# B&R Automation Studio project EFI (part 17)

### LineCtrl.typ
```iecst
TYPE
	LineControlAlarms_typ : 	STRUCT
		xAlrOvervoltage : BOOL; (*Warning alarm*)
		xAlrPrinterNoPowered : BOOL; (*Warning alarm*)
		xAlr24VdcStartSeqNoPowered : BOOL; (*Warning alarm*)
		xResetCondition : BOOL;
		xStopAlarm : BOOL;
		xCriticalAlarm : BOOL;
		xWarningAlarm : BOOL;
		xAlarmNonReseteable : BOOL;
		xAlarmReseteable : BOOL;
		xAlarmSound : BOOL;
		iReasonStop : UDINT; (*The reason to move the machine to stop*)
		iReasonWarning : UDINT;
		iReasonResetCondition : UDINT; (*The reason to active light tower's blue light*)
		iReasonCritical : UDINT; (*The reason to move the machine out of auto mode*)
	END_STRUCT;
	LineControlCommands_typ : 	STRUCT
		CalibrateCamera : BOOL;
		Print : BOOL; (*Edge commands. Reseted when managed*)
		Pause : BOOL; (*Edge commands. Reseted when managed*)
		ControlStop : BOOL; (*Edge commands. Reseted when managed*)
		Stop : BOOL; (*Edge commands. Reseted when managed*)
		Clean : BOOL; (*Edge commands. Reseted when managed*)
		EmptyBelt : BOOL; (*Edge commands. Reseted when managed*)
		PowerOff : BOOL;
		StartUp : StartUpCommands_typ;
	END_STRUCT;
	LineControlParameters_typ : 	STRUCT
		ExternalDevices : ARRAY[0..MAX_EXTERNAL_DEVICES]OF StartUpParameters_typ; (*0:Feeder||1:Primer||2:Printer||3:Dryer1||4:Dryer2||5:DryerCtrl||6:Stacker||7:UV||8:Chiller||9:Hoopers||10:OPV*)
		iNumExternalDevices : INT := 0;
		iLightTowerMode : INT; (*0: IEC Standard, 1: Customer1 request, 2: Customer2 request*)
		xBatchFeeding : BOOL; (*1: Batch feeding, 0: Continous feeding*)
		Hw : LineControlHwParameters_typ;
	END_STRUCT;
	LineControlInputs_typ : 	STRUCT
		xOvervoltageProtectionOk : BOOL;
		xPrinterPowered : BOOL;
		x24VdcStartSeqNoPowered : BOOL;
		UPSs : ARRAY[0..2]OF UPS_Inputs;
		Customer : ARRAY[0..3]OF BOOL;
	END_STRUCT;
	StartUpInputs_typ : 	STRUCT
		xPowered : BOOL; (*Some devices power management needs a second signal to switch off its branch*)
	END_STRUCT;
	StartUpOutputs_typ : 	STRUCT
		xClose : BOOL; (*Signal to active contactor coil of device's power branch*)
		xOpen : BOOL; (*Before activating the Close signal, the Open output has to be activated. A NC signal through a relay is sent as Open, so just sending close both signals are electrically sent*)
	END_STRUCT;
	LineControlOutputs_typ : 	STRUCT
		ExternalDevices : ARRAY[0..MAX_EXTERNAL_DEVICES]OF StartUpOutputs_typ; (*Signal to active contactor coil of device's power branch*)
		xRedLight : BOOL;
		xYellowLight : BOOL;
		xGreenLight : BOOL;
		xWhiteLight : BOOL;
		xBlueLight : BOOL;
		xLightReset : BOOL;
		xSound : BOOL;
		Customer : ARRAY[0..3]OF BOOL;
		Sw : LineControlOutputsForSw;
	END_STRUCT;
	StartUpCommands_typ : 	STRUCT
		xPowerOff : ARRAY[0..MAX_EXTERNAL_DEVICES]OF BOOL; (*0:Feeder||1:Primer||2:Printer||3:Dryer1||4:Dryer2||5:DryerCtrl||6:Stacker||7:UV||8:Chiller||9:Hoopers||10:OPV*)
		xPowerUp : ARRAY[0..MAX_EXTERNAL_DEVICES]OF BOOL; (*0:Feeder||1:Primer||2:Printer||3:Dryer1||4:Dryer2||5:DryerCtrl||6:Stacker||7:UV||8:Chiller||9:Hoopers||10:OPV*)
		xStartAll : BOOL;
	END_STRUCT;
	StartUpParameters_typ : 	STRUCT
		tiDelay : TIME; (*Delay to activate from the previous device*)
		xIsEngine : BOOL; (*Activate if the Power is set to de Device through a Motorized contactor*)
	END_STRUCT;
	LineControl_typ : 	STRUCT
		Commands : LineControlCommands_typ;
		Status : LineStatus_enum := LINE_NOT_POWERED;
		StatusSw : UINT := 0; (*Copy for Sw*)
		Alarms : LineControlAlarms_typ;
		Parameters : LineControlParameters_typ;
		Outputs : LineControlOutputs_typ;
		Inputs : LineControlInputs_typ;
		SubStatus : UINT; (*Substatus of Line.Status. Info useful for reports and debug*)
		StatusSummary : LineControlStatusSummarized; (*Struct to summarize different states that belongs to same process*)
		OrdersSw : LineControlOrdersSw_typ;
		Orders : LineControlOrders_typ;
	END_STRUCT;
	LineControlOutputsForSw : 	STRUCT
		xPrintOrderRequestToSw : BOOL;
		xCleanOrderRequestToSw : BOOL;
		iTimesBlockAtSafePosition : UINT; (*Counter to acknowledge how many times block has been lifted to safe position*)
	END_STRUCT;
	LineControlOrders_typ : 	STRUCT
		Preprinting : BOOL; (*Order to the printer to go to preprint position*)
	END_STRUCT;
	LineControlOrdersSw_typ : 	STRUCT
		Shutdown : BOOL;
	END_STRUCT;
	LineControlHwParameters_typ : 	STRUCT
		rMaxSpeed : REAL; (*Speed in mm/min*)
		xDoubleLineAllowed : BOOL; (*Active when allows double line printing*)
	END_STRUCT;
END_TYPE
```

### Library Logical/LineCtrl/LineCtrl

#### LineCtrlFunctions.fun
```iecst
{REDUND_ERROR} FUNCTION CuringSystemsStarted : BOOL (*TODO: Add your comment here*) (*$GROUP=User,$CAT=User,$GROUPICON=User.png,$CATICON=User.png*)
	VAR_INPUT
		CuringLed : REFERENCE TO CuringLed_typ;
	END_VAR
END_FUNCTION

{REDUND_ERROR} FUNCTION CuringSystemsReady : BOOL (*TODO: Add your comment here*) (*$GROUP=User,$CAT=User,$GROUPICON=User.png,$CATICON=User.png*)
	VAR_INPUT
		CuringLed : REFERENCE TO CuringLed_typ;
	END_VAR
END_FUNCTION

{REDUND_ERROR} FUNCTION PrinterBeltStopped : BOOL (*TODO: Add your comment here*) (*$GROUP=User,$CAT=User,$GROUPICON=User.png,$CATICON=User.png*)
	VAR_INPUT
		Belt : REFERENCE TO stBelt;
	END_VAR
END_FUNCTION

{REDUND_ERROR} FUNCTION PrinterBeltStarted : BOOL (*TODO: Add your comment here*) (*$GROUP=User,$CAT=User,$GROUPICON=User.png,$CATICON=User.png*)
	VAR_INPUT
		Belt : REFERENCE TO stBelt;
	END_VAR
END_FUNCTION

{REDUND_ERROR} FUNCTION DryerReady : BOOL (*TODO: Add your comment here*) (*$GROUP=User,$CAT=User,$GROUPICON=User.png,$CATICON=User.png*)
	VAR_INPUT
		Dryer : REFERENCE TO DryerAnc_typ;
	END_VAR
END_FUNCTION

{REDUND_ERROR} FUNCTION FeederReady : BOOL (*TODO: Add your comment here*) (*$GROUP=User,$CAT=User,$GROUPICON=User.png,$CATICON=User.png*)
	VAR_INPUT
		Feeder : REFERENCE TO Feeder_typ;
	END_VAR
END_FUNCTION

{REDUND_ERROR} FUNCTION PrimerReady : BOOL (*TODO: Add your comment here*) (*$GROUP=User,$CAT=User,$GROUPICON=User.png,$CATICON=User.png*)
	VAR_INPUT
		Primer : REFERENCE TO Primer_typ;
	END_VAR
END_FUNCTION

{REDUND_ERROR} FUNCTION SarmStopped : BOOL (*TODO: Add your comment here*) (*$GROUP=User,$CAT=User,$GROUPICON=User.png,$CATICON=User.png*)
	VAR_INPUT
		Sarm : REFERENCE TO Sarm_typ;
	END_VAR
END_FUNCTION

{REDUND_ERROR} FUNCTION SarmStarted : BOOL (*TODO: Add your comment here*) (*$GROUP=User,$CAT=User,$GROUPICON=User.png,$CATICON=User.png*)
	VAR_INPUT
		Sarm : REFERENCE TO Sarm_typ;
	END_VAR
END_FUNCTION

{REDUND_ERROR} FUNCTION SarmReady : BOOL (*TODO: Add your comment here*) (*$GROUP=User,$CAT=User,$GROUPICON=User.png,$CATICON=User.png*)
	VAR_INPUT
		Sarm : REFERENCE TO Sarm_typ;
	END_VAR
END_FUNCTION

FUNCTION EhdAdjusted : BOOL
	VAR_INPUT
		EdgeHoldDown : REFERENCE TO EdgeHoldDown_typ;
	END_VAR
END_FUNCTION

FUNCTION EhdReady : BOOL
	VAR_INPUT
		EdgeHoldDown : REFERENCE TO EdgeHoldDown_typ;
	END_VAR
END_FUNCTION

{REDUND_ERROR} FUNCTION StackerReady : BOOL (*TODO: Add your comment here*) (*$GROUP=User,$CAT=User,$GROUPICON=User.png,$CATICON=User.png*)
	VAR_INPUT
		Stacker : REFERENCE TO Stacker_typ;
	END_VAR
END_FUNCTION

{REDUND_ERROR} FUNCTION BarPositionCleaning : BOOL (*TODO: Add your comment here*) (*$GROUP=User,$CAT=User,$GROUPICON=User.png,$CATICON=User.png*)
	VAR_INPUT
		Machine : REFERENCE TO StGeneral;
	END_VAR
END_FUNCTION

{REDUND_ERROR} FUNCTION BarPositionCapped : BOOL (*TODO: Add your comment here*) (*$GROUP=User,$CAT=User,$GROUPICON=User.png,$CATICON=User.png*)
	VAR_INPUT
		Machine : REFERENCE TO StGeneral;
	END_VAR
END_FUNCTION

{REDUND_ERROR} FUNCTION JobReady : BOOL (*TODO: Add your comment here*) (*$GROUP=User,$CAT=User,$GROUPICON=User.png,$CATICON=User.png*)
	VAR_INPUT
		Machine : REFERENCE TO StGeneral;
	END_VAR
END_FUNCTION

{REDUND_ERROR} FUNCTION BarPositionReady : BOOL (*TODO: Add your comment here*) (*$GROUP=User,$CAT=User,$GROUPICON=User.png,$CATICON=User.png*)
	VAR_INPUT
		Machine : REFERENCE TO StGeneral;
	END_VAR
END_FUNCTION

{REDUND_ERROR} FUNCTION DryerStarted : BOOL (*TODO: Add your comment here*) (*$GROUP=User,$CAT=User,$GROUPICON=User.png,$CATICON=User.png*)
	VAR_INPUT
		Dryer : REFERENCE TO DryerAnc_typ;
	END_VAR
END_FUNCTION

{REDUND_ERROR} FUNCTION FeederStarted : BOOL (*TODO: Add your comment here*) (*$GROUP=User,$CAT=User,$GROUPICON=User.png,$CATICON=User.png*)
	VAR_INPUT
		Feeder : REFERENCE TO Feeder_typ;
	END_VAR
END_FUNCTION

{REDUND_ERROR} FUNCTION PrimerStarted : BOOL (*TODO: Add your comment here*) (*$GROUP=User,$CAT=User,$GROUPICON=User.png,$CATICON=User.png*)
	VAR_INPUT
		Primer : REFERENCE TO Primer_typ;
	END_VAR
END_FUNCTION

{REDUND_ERROR} FUNCTION StackerStarted : BOOL (*TODO: Add your comment here*) (*$GROUP=User,$CAT=User,$GROUPICON=User.png,$CATICON=User.png*)
	VAR_INPUT
		Stacker : REFERENCE TO Stacker_typ;
	END_VAR
END_FUNCTION

{REDUND_ERROR} FUNCTION ThicknessSensorReady : BOOL (*TODO: Add your comment here*) (*$GROUP=User,$CAT=User,$GROUPICON=User.png,$CATICON=User.png*)
	VAR_INPUT
		ThickCtrl : REFERENCE TO stThicknessCtrl_typ;
	END_VAR
END_FUNCTION

{REDUND_ERROR} FUNCTION DryerPaused : BOOL (*TODO: Add your comment here*) (*$GROUP=User,$CAT=User,$GROUPICON=User.png,$CATICON=User.png*)
	VAR_INPUT
		Dryer : REFERENCE TO DryerAnc_typ;
	END_VAR
END_FUNCTION

{REDUND_ERROR} FUNCTION PrimerPaused : BOOL (*TODO: Add your comment here*) (*$GROUP=User,$CAT=User,$GROUPICON=User.png,$CATICON=User.png*)
	VAR_INPUT
		Primer : REFERENCE TO Primer_typ;
	END_VAR
END_FUNCTION

{REDUND_ERROR} FUNCTION FeederPaused : BOOL (*TODO: Add your comment here*) (*$GROUP=User,$CAT=User,$GROUPICON=User.png,$CATICON=User.png*)
	VAR_INPUT
		Feeder : REFERENCE TO Feeder_typ;
	END_VAR
END_FUNCTION

{REDUND_ERROR} FUNCTION DryerStopped : BOOL (*TODO: Add your comment here*) (*$GROUP=User,$CAT=User,$GROUPICON=User.png,$CATICON=User.png*)
	VAR_INPUT
		Dryer : REFERENCE TO DryerAnc_typ;
	END_VAR
END_FUNCTION

{REDUND_ERROR} FUNCTION FeederStopped : BOOL (*TODO: Add your comment here*) (*$GROUP=User,$CAT=User,$GROUPICON=User.png,$CATICON=User.png*)
	VAR_INPUT
		Feeder : REFERENCE TO Feeder_typ;
	END_VAR
END_FUNCTION

{REDUND_ERROR} FUNCTION PrimerStopped : BOOL (*TODO: Add your comment here*) (*$GROUP=User,$CAT=User,$GROUPICON=User.png,$CATICON=User.png*)
	VAR_INPUT
		Primer : REFERENCE TO Primer_typ;
	END_VAR
END_FUNCTION

{REDUND_ERROR} FUNCTION StackerStopped : BOOL (*TODO: Add your comment here*) (*$GROUP=User,$CAT=User,$GROUPICON=User.png,$CATICON=User.png*)
	VAR_INPUT
		Stacker : REFERENCE TO Stacker_typ;
	END_VAR
END_FUNCTION

FUNCTION EhdStopped : BOOL
	VAR_INPUT
		EdgeHoldDown : REFERENCE TO EdgeHoldDown_typ;
	END_VAR
END_FUNCTION

{REDUND_ERROR} FUNCTION FeederNotFeeding : BOOL (*TODO: Add your comment here*) (*$GROUP=User,$CAT=User,$GROUPICON=User.png,$CATICON=User.png*)
	VAR_INPUT
		Feeder : REFERENCE TO Feeder_typ;
	END_VAR
END_FUNCTION

{REDUND_ERROR} FUNCTION OpvReady : BOOL (*TODO: Add your comment here*) (*$GROUP=User,$CAT=User,$GROUPICON=User.png,$CATICON=User.png*)
	VAR_INPUT
		OverVarnish : REFERENCE TO Opv_typ;
	END_VAR
END_FUNCTION

{REDUND_ERROR} FUNCTION OpvStarted : BOOL (*TODO: Add your comment here*) (*$GROUP=User,$CAT=User,$GROUPICON=User.png,$CATICON=User.png*)
	VAR_INPUT
		OverVarnish : REFERENCE TO Opv_typ;
	END_VAR
END_FUNCTION

FUNCTION SarmPaused : BOOL
	VAR_INPUT
		Sarm : REFERENCE TO Sarm_typ;
	END_VAR
END_FUNCTION

{REDUND_ERROR} FUNCTION OpvPaused : BOOL (*TODO: Add your comment here*) (*$GROUP=User,$CAT=User,$GROUPICON=User.png,$CATICON=User.png*)
	VAR_INPUT
		OverVarnish : REFERENCE TO Opv_typ;
	END_VAR
END_FUNCTION

{REDUND_ERROR} FUNCTION OpvStopped : BOOL (*TODO: Add your comment here*) (*$GROUP=User,$CAT=User,$GROUPICON=User.png,$CATICON=User.png*)
	VAR_INPUT
		OverVarnish : REFERENCE TO Opv_typ;
	END_VAR
END_FUNCTION

{REDUND_ERROR} FUNCTION FeederEmptied : BOOL (*TODO: Add your comment here*) (*$GROUP=User,$CAT=User,$GROUPICON=User.png,$CATICON=User.png*)
	VAR_INPUT
		Feeder : REFERENCE TO Feeder_typ;
	END_VAR
END_FUNCTION

{REDUND_ERROR} FUNCTION StackerEmptied : BOOL (*TODO: Add your comment here*) (*$GROUP=User,$CAT=User,$GROUPICON=User.png,$CATICON=User.png*)
	VAR_INPUT
		Stacker : REFERENCE TO Stacker_typ;
	END_VAR
END_FUNCTION

{REDUND_ERROR} FUNCTION OpvEmptied : BOOL (*TODO: Add your comment here*) (*$GROUP=User,$CAT=User,$GROUPICON=User.png,$CATICON=User.png*)
	VAR_INPUT
		OverVarnish : REFERENCE TO Opv_typ;
	END_VAR
END_FUNCTION

{REDUND_ERROR} FUNCTION DryerEmptied : BOOL (*TODO: Add your comment here*) (*$GROUP=User,$CAT=User,$GROUPICON=User.png,$CATICON=User.png*)
	VAR_INPUT
		Dryer : REFERENCE TO DryerAnc_typ;
	END_VAR
END_FUNCTION

{REDUND_ERROR} FUNCTION PrinterEmptied : BOOL (*TODO: Add your comment here*) (*$GROUP=User,$CAT=User,$GROUPICON=User.png,$CATICON=User.png*)
	VAR_INPUT
		ThickCtrl : REFERENCE TO stThicknessCtrl_typ;
	END_VAR
END_FUNCTION

{REDUND_ERROR} FUNCTION PrimerEmptied : BOOL (*TODO: Add your comment here*) (*$GROUP=User,$CAT=User,$GROUPICON=User.png,$CATICON=User.png*)
	VAR_INPUT
		Primer : REFERENCE TO Primer_typ;
	END_VAR
END_FUNCTION

FUNCTION SarmEmptied : BOOL
	VAR_INPUT
		Sarm : REFERENCE TO Sarm_typ;
	END_VAR
END_FUNCTION

{REDUND_ERROR} FUNCTION DryerMaxSpeed : REAL (*TODO: Add your comment here*) (*$GROUP=User,$CAT=User,$GROUPICON=User.png,$CATICON=User.png*)
	VAR_INPUT
		Dryer : REFERENCE TO DryerAnc_typ;
		Belt : REFERENCE TO stBelt;
	END_VAR
END_FUNCTION

{REDUND_ERROR} FUNCTION DryerMaxMediaLength : UINT (*TODO: Add your comment here*) (*$GROUP=User,$CAT=User,$GROUPICON=User.png,$CATICON=User.png*)
	VAR_INPUT
		Dryer : REFERENCE TO DryerAnc_typ;
		Machine : REFERENCE TO StGeneral;
	END_VAR
END_FUNCTION

{REDUND_ERROR} FUNCTION DryerMaxMediaWidth : UINT (*TODO: Add your comment here*) (*$GROUP=User,$CAT=User,$GROUPICON=User.png,$CATICON=User.png*)
	VAR_INPUT
		Dryer : REFERENCE TO DryerAnc_typ;
		Machine : REFERENCE TO StGeneral;
	END_VAR
END_FUNCTION

{REDUND_ERROR} FUNCTION FeederMaxSpeed : REAL (*TODO: Add your comment here*) (*$GROUP=User,$CAT=User,$GROUPICON=User.png,$CATICON=User.png*)
	VAR_INPUT
		Feeder : REFERENCE TO Feeder_typ;
		Belt : REFERENCE TO stBelt;
	END_VAR
END_FUNCTION

{REDUND_ERROR} FUNCTION FeederMaxMediaThickness : UINT (*TODO: Add your comment here*) (*$GROUP=User,$CAT=User,$GROUPICON=User.png,$CATICON=User.png*)
	VAR_INPUT
		Feeder : REFERENCE TO Feeder_typ;
		Machine : REFERENCE TO StGeneral;
	END_VAR
END_FUNCTION

{REDUND_ERROR} FUNCTION FeederMinMediaThickness : UINT (*TODO: Add your comment here*) (*$GROUP=User,$CAT=User,$GROUPICON=User.png,$CATICON=User.png*)
	VAR_INPUT
		Feeder : REFERENCE TO Feeder_typ;
		Machine : REFERENCE TO StGeneral;
	END_VAR
END_FUNCTION

{REDUND_ERROR} FUNCTION FeederMaxMediaLength : UINT (*TODO: Add your comment here*) (*$GROUP=User,$CAT=User,$GROUPICON=User.png,$CATICON=User.png*)
	VAR_INPUT
		Feeder : REFERENCE TO Feeder_typ;
		Machine : REFERENCE TO StGeneral;
	END_VAR
END_FUNCTION

{REDUND_ERROR} FUNCTION FeederMaxMediaWidth : UINT (*TODO: Add your comment here*) (*$GROUP=User,$CAT=User,$GROUPICON=User.png,$CATICON=User.png*)
	VAR_INPUT
		Feeder : REFERENCE TO Feeder_typ;
		Machine : REFERENCE TO StGeneral;
	END_VAR
END_FUNCTION

{REDUND_ERROR} FUNCTION PrimerMaxSpeed : REAL (*TODO: Add your comment here*) (*$GROUP=User,$CAT=User,$GROUPICON=User.png,$CATICON=User.png*)
	VAR_INPUT
		Primer : REFERENCE TO Primer_typ;
		Belt : REFERENCE TO stBelt;
	END_VAR
END_FUNCTION

{REDUND_ERROR} FUNCTION PrimerMinMediaThickness : UINT (*TODO: Add your comment here*) (*$GROUP=User,$CAT=User,$GROUPICON=User.png,$CATICON=User.png*)
	VAR_INPUT
		Primer : REFERENCE TO Primer_typ;
		Machine : REFERENCE TO StGeneral;
	END_VAR
END_FUNCTION

{REDUND_ERROR} FUNCTION PrimerMaxMediaThickness : UINT (*TODO: Add your comment here*) (*$GROUP=User,$CAT=User,$GROUPICON=User.png,$CATICON=User.png*)
	VAR_INPUT
		Primer : REFERENCE TO Primer_typ;
		Machine : REFERENCE TO StGeneral;
	END_VAR
END_FUNCTION

{REDUND_ERROR} FUNCTION PrimerMaxMediaLength : UINT (*TODO: Add your comment here*) (*$GROUP=User,$CAT=User,$GROUPICON=User.png,$CATICON=User.png*)
	VAR_INPUT
		Primer : REFERENCE TO Primer_typ;
		Machine : REFERENCE TO StGeneral;
	END_VAR
END_FUNCTION

{REDUND_ERROR} FUNCTION PrimerMaxMediaWidth : UINT (*TODO: Add your comment here*) (*$GROUP=User,$CAT=User,$GROUPICON=User.png,$CATICON=User.png*)
	VAR_INPUT
		Primer : REFERENCE TO Primer_typ;
		Machine : REFERENCE TO StGeneral;
	END_VAR
END_FUNCTION

{REDUND_ERROR} FUNCTION OvervarnishMaxSpeed : REAL (*TODO: Add your comment here*) (*$GROUP=User,$CAT=User,$GROUPICON=User.png,$CATICON=User.png*)
	VAR_INPUT
		OverVarnish : REFERENCE TO Opv_typ;
		Belt : REFERENCE TO stBelt;
	END_VAR
END_FUNCTION

{REDUND_ERROR} FUNCTION OvervarnishMaxMediaLength : UINT (*TODO: Add your comment here*) (*$GROUP=User,$CAT=User,$GROUPICON=User.png,$CATICON=User.png*)
	VAR_INPUT
		OverVarnish : REFERENCE TO Opv_typ;
		Machine : REFERENCE TO StGeneral;
	END_VAR
END_FUNCTION

{REDUND_ERROR} FUNCTION OverVarnishMaxMediaThickness : UINT (*TODO: Add your comment here*) (*$GROUP=User,$CAT=User,$GROUPICON=User.png,$CATICON=User.png*)
	VAR_INPUT
		OverVarnish : REFERENCE TO Opv_typ;
		Machine : REFERENCE TO StGeneral;
	END_VAR
END_FUNCTION

{REDUND_ERROR} FUNCTION OverVarnishMinMediaThickness : UINT (*TODO: Add your comment here*) (*$GROUP=User,$CAT=User,$GROUPICON=User.png,$CATICON=User.png*)
	VAR_INPUT
		OverVarnish : REFERENCE TO Opv_typ;
		Machine : REFERENCE TO StGeneral;
	END_VAR
END_FUNCTION

{REDUND_ERROR} FUNCTION OvervarnishMaxMediaWidth : UINT (*TODO: Add your comment here*) (*$GROUP=User,$CAT=User,$GROUPICON=User.png,$CATICON=User.png*)
	VAR_INPUT
		OverVarnish : REFERENCE TO Opv_typ;
		Machine : REFERENCE TO StGeneral;
	END_VAR
END_FUNCTION

{REDUND_ERROR} FUNCTION StackerMaxSpeed : REAL (*TODO: Add your comment here*) (*$GROUP=User,$CAT=User,$GROUPICON=User.png,$CATICON=User.png*)
	VAR_INPUT
		Stacker : REFERENCE TO Stacker_typ;
		Belt : REFERENCE TO stBelt;
	END_VAR
END_FUNCTION

{REDUND_ERROR} FUNCTION StackerMaxMediaLength : UINT (*TODO: Add your comment here*) (*$GROUP=User,$CAT=User,$GROUPICON=User.png,$CATICON=User.png*)
	VAR_INPUT
		Stacker : REFERENCE TO Stacker_typ;
		Machine : REFERENCE TO StGeneral;
	END_VAR
END_FUNCTION

{REDUND_ERROR} FUNCTION StackerMaxMediaThickness : UINT (*TODO: Add your comment here*) (*$GROUP=User,$CAT=User,$GROUPICON=User.png,$CATICON=User.png*)
	VAR_INPUT
		Stacker : REFERENCE TO Stacker_typ;
		Machine : REFERENCE TO StGeneral;
	END_VAR
END_FUNCTION

{REDUND_ERROR} FUNCTION StackerMinMediaThickness : UINT (*TODO: Add your comment here*) (*$GROUP=User,$CAT=User,$GROUPICON=User.png,$CATICON=User.png*)
	VAR_INPUT
		Stacker : REFERENCE TO Stacker_typ;
		Machine : REFERENCE TO StGeneral;
	END_VAR
END_FUNCTION

{REDUND_ERROR} FUNCTION StackerMaxMediaWidth : UINT (*TODO: Add your comment here*) (*$GROUP=User,$CAT=User,$GROUPICON=User.png,$CATICON=User.png*)
	VAR_INPUT
		Stacker : REFERENCE TO Stacker_typ;
		Machine : REFERENCE TO StGeneral;
	END_VAR
END_FUNCTION

{REDUND_ERROR} FUNCTION SarmMaxSpeed : REAL (*TODO: Add your comment here*) (*$GROUP=User,$CAT=User,$GROUPICON=User.png,$CATICON=User.png*)
	VAR_INPUT
		Sarm : REFERENCE TO Sarm_typ;
		Belt : REFERENCE TO stBelt;
	END_VAR
END_FUNCTION

{REDUND_ERROR} FUNCTION SarmMaxMediaThickness : UINT (*TODO: Add your comment here*) (*$GROUP=User,$CAT=User,$GROUPICON=User.png,$CATICON=User.png*)
	VAR_INPUT
		Sarm : REFERENCE TO Sarm_typ;
		Machine : REFERENCE TO StGeneral;
	END_VAR
END_FUNCTION

{REDUND_ERROR} FUNCTION SarmMinMediaThickness : UINT (*TODO: Add your comment here*) (*$GROUP=User,$CAT=User,$GROUPICON=User.png,$CATICON=User.png*)
	VAR_INPUT
		Sarm : REFERENCE TO Sarm_typ;
		Machine : REFERENCE TO StGeneral;
	END_VAR
END_FUNCTION

{REDUND_ERROR} FUNCTION SarmMaxMediaLength : UINT (*TODO: Add your comment here*) (*$GROUP=User,$CAT=User,$GROUPICON=User.png,$CATICON=User.png*)
	VAR_INPUT
		Sarm : REFERENCE TO Sarm_typ;
		Machine : REFERENCE TO StGeneral;
	END_VAR
END_FUNCTION

{REDUND_ERROR} FUNCTION SarmMaxMediaWidth : UINT (*TODO: Add your comment here*) (*$GROUP=User,$CAT=User,$GROUPICON=User.png,$CATICON=User.png*)
	VAR_INPUT
		Sarm : REFERENCE TO Sarm_typ;
		Machine : REFERENCE TO StGeneral;
	END_VAR
END_FUNCTION
```

#### CleaningBelt.st
```iecst
ACTION CleaningBelt:
	IF xStatusChanged THEN
		iLineStatus:=720;
	END_IF

	CASE iLineStatus OF
		720:
			gMachine.commands.CleanBelt.xStart := FALSE;
			xCleanBeltToBeExecuted := FALSE;
			IF gBeltClean.Status.State = BCLEAN_FAULT OR NOT gMachine.St.Position.xCleaning AND NOT BeltClean.Status.xCleaning THEN
				IF xPreviousIdle THEN
					gMachine.commands.xRunBelt := FALSE;
				END_IF
				xLineReady:=TRUE;
			END_IF
	END_CASE

END_ACTION
```

#### ControlStopping.st
```iecst
ACTION ControlStopping:

	IF xStatusChanged THEN
		ton_PrinterBeltInputEmpty.IN := FALSE;
		iLineStatus:=500;
	END_IF

	ton_PrinterBeltInputEmpty();

	CASE iLineStatus OF

		500:
			gMachine.commands.xClean:=FALSE;

			IF gMachine.AlSummary.xAlarmStop THEN
				Feeder.Commands.xStop:=TRUE;
				Primer.Commands.xStop:=TRUE;
				Sarm.Commands.xStop:=TRUE;
				gMachine.commands.xStop:=TRUE;
				gMachine.commands.xRunBelt:=FALSE; //This shouldnt be required, Why stop command does not stop the belt?
				StopCuringSystems;
				StopBlowers;
				iLineStatus:=506;

			ELSIF Sarm.Alarms.xCriticalAlarm THEN
				Feeder.Commands.xStop:=TRUE;
				Primer.Commands.xStop:=TRUE;
				Sarm.Commands.xStop:=TRUE;
				iLineStatus:=504;

			ELSIF Primer.Alarms.xCriticalAlarm THEN
				Feeder.Commands.xStop:=TRUE;
				Primer.Commands.xStop:=TRUE;

				iLineStatus:=503;
			ELSE
				iLineStatus:=iLineStatus+1;
			END_IF

		501:
			Feeder.Commands.xStop:=TRUE;
			iLineStatus:=iLineStatus+1;

		502:
			xFeederNotFeeding := FeederNotFeeding(ADR(Feeder));
			IF xFeederNotFeeding THEN
				Primer.Commands.xControlStop:=TRUE;
				iLineStatus:=iLineStatus+1;
			END_IF

			IF gMachine.AlSummary.xAlarmStop THEN
				Feeder.Commands.xStop:=TRUE;
				Primer.Commands.xStop:=TRUE;
				Sarm.Commands.xStop:=TRUE;
				gMachine.commands.xStop:=TRUE;
				gMachine.commands.xRunBelt:=FALSE; //This shouldnt be required, Why stop command does not stop the belt?
				StopCuringSystems;
				StopBlowers;
				iLineStatus:=506;

			ELSIF Sarm.Alarms.xCriticalAlarm THEN
				Feeder.Commands.xStop:=TRUE;
				Primer.Commands.xStop:=TRUE;
				Sarm.Commands.xStop:=TRUE;
				iLineStatus:=504;

			ELSIF Primer.Alarms.xCriticalAlarm THEN
				Feeder.Commands.xStop:=TRUE;
				Primer.Commands.xStop:=TRUE;

				iLineStatus:=503;
			END_IF

		503:
			xPrimerStopped := PrimerStopped(ADR(Primer));
			IF xPrimerStopped THEN
				Sarm.Commands.xControlStop:=TRUE;
				iLineStatus:=iLineStatus+1;
			END_IF

			IF gMachine.AlSummary.xAlarmStop THEN
				Feeder.Commands.xStop:=TRUE;
				Primer.Commands.xStop:=TRUE;
				Sarm.Commands.xStop:=TRUE;
				gMachine.commands.xStop:=TRUE;
				gMachine.commands.xRunBelt:=FALSE; //This shouldnt be required, Why stop command does not stop the belt?
				StopCuringSystems;
				StopBlowers;
				iLineStatus:=506;

			ELSIF Sarm.Alarms.xCriticalAlarm THEN
				Feeder.Commands.xStop:=TRUE;
				Primer.Commands.xStop:=TRUE;
				Sarm.Commands.xStop:=TRUE;
				iLineStatus:=504;
			END_IF

		504:
			xSarmStopped := SarmStopped(ADR(Sarm));
			IF xSarmStopped THEN
				iLineStatus:=iLineStatus+1;
			END_IF

			IF gMachine.AlSummary.xAlarmStop THEN
				Feeder.Commands.xStop:=TRUE;
				Primer.Commands.xStop:=TRUE;
				Sarm.Commands.xStop:=TRUE;
				gMachine.commands.xStop:=TRUE;
				gMachine.commands.xRunBelt:=FALSE; //This shouldnt be required, Why stop command does not stop the belt?
				StopCuringSystems;
				StopBlowers;
				iLineStatus:=506;
			END_IF

		505:
			//Timer
			tiTimeToEmpty := REAL_TO_TIME(60 * (gMachine.Pt.CT.rDistanceBeltInitToPd) / Belt.parameters.rSetPointSpeed); //Belt.parameters.rSetPointSpeed minimum value is 5m/min, cannot be 0.
			ton_PrinterBeltInputEmpty.IN := TRUE;
			ton_PrinterBeltInputEmpty.PT := tiTimeToEmpty;

			xPrinterBeltInputEmpty := ton_PrinterBeltInputEmpty.Q;

			xPrinterBeltStopped:= PrinterBeltStopped(ADR(Belt));
			IF (xPrinterBeltInputEmpty OR xFromPause) AND (xPrinterEmptied OR xPrinterBeltStopped) THEN
				StopCuringSystems;
				StopBlowers;

				EdgeHoldDown.commands.xStop := TRUE;

				iLineStatus:=iLineStatus+1;
			END_IF

			IF gMachine.AlSummary.xAlarmStop THEN
				Feeder.Commands.xStop:=TRUE;
				Primer.Commands.xStop:=TRUE;
				Sarm.Commands.xStop:=TRUE;
				gMachine.commands.xStop:=TRUE;
				gMachine.commands.xRunBelt:=FALSE; //This shouldnt be required, Why stop command does not stop the belt?
				StopCuringSystems;
				StopBlowers;
				iLineStatus:=506;
			END_IF

		506:
			xEhdStopped := EhdStopped(ADR(EdgeHoldDown));
			IF xEhdStopped AND xDryerEmptied AND xOpvEmptied THEN
				gMachine.commands.xStop:=TRUE;
				gMachine.commands.xRunBelt:=FALSE;

				EdgeHoldDown.orders.xAdjustToMedia:=FALSE;
				EdgeHoldDown.orders.xResetPosition:=TRUE;

				Dryer.Commands.xControlStop:=TRUE;
				iLineStatus:=iLineStatus+1;
			END_IF

		507:
			xDryerStopped := DryerStopped(ADR(Dryer));
			IF xDryerStopped THEN
				OverVarnish.Commands.xControlStop:=TRUE;
				iLineStatus:=iLineStatus+1;
			END_IF

		508:
			xOverVarnishStopped := OpvStopped(ADR(OverVarnish));
			IF xOverVarnishStopped THEN
				Stacker.Commands.xControlStop:=TRUE;
				iLineStatus:=iLineStatus+1;
			END_IF

		509:
			xBarsInCapPosition := BarPositionCapped(ADR(Machine));
			xEhdReady := EhdReady(ADR(EdgeHoldDown));
			IF xEhdReady AND xBarsInCapPosition THEN
				iLineStatus:=iLineStatus+1;
			END_IF

		510:
			xStackerStopped := StackerStopped(ADR(Stacker));
			IF xStackerStopped THEN
				xLineReady:=TRUE;
			END_IF

	END_CASE

END_ACTION

ACTION StopCuringSystems:

END_ACTION

ACTION StopBlowers:
	FOR iIndexTransVacuum:=1 TO MAX_LAST_TRANS_VACUUM DO
		TransVacuum[iIndexTransVacuum].Commands.xRunByLine := FALSE;
	END_FOR
END_ACTION
```

#### EmptyingBelt.st
```iecst
ACTION EmptyingBelt:

	IF xStatusChanged THEN
		ton_PrinterBeltInputEmpty.IN := FALSE;
		iLineStatus:=220;
	END_IF

	//DELOREAN-830:To lift bars up when there are no printed boards below bars, so no more curing is required
	IF (NOT ThickCtrl.status.MediaPosition.xMediaBelowMachine) THEN gMachine.commands.xAllToCap:=TRUE; END_IF

	ton_PrinterBeltInputEmpty();

	CASE iLineStatus OF
		220:
			IF xFeederEmptied THEN
				Feeder.Commands.xStop := TRUE;
				iLineStatus:=iLineStatus+1;
			END_IF

		221:
			IF xPrimerEmptied THEN
				Primer.Commands.xControlStop:=TRUE;
				iLineStatus:=iLineStatus+1;
			END_IF

		222:
			IF xSarmEmptied THEN
				Sarm.Commands.xControlStop := TRUE;
				iLineStatus:=iLineStatus+1;
			END_IF

		223:
			//Timer
			tiTimeToEmpty := REAL_TO_TIME(60 * (UINT_TO_REAL (gThicknessCtrl.parameters.Belt.iBeltPerimeterLength * 5)) / Belt.parameters.rSetPointSpeed); //Belt.parameters.rSetPointSpeed minimum value is 5m/min, cannot be 0.
			ton_PrinterBeltInputEmpty.IN := TRUE;
			ton_PrinterBeltInputEmpty.PT := tiTimeToEmpty;

			xPrinterBeltInputEmpty := ton_PrinterBeltInputEmpty.Q;
			IF xPrinterEmptied AND xPrinterBeltInputEmpty THEN
				iLineStatus:=iLineStatus+1;
			END_IF

		224:
			IF xDryerEmptied THEN
				iLineStatus:=iLineStatus+1;
			END_IF

		225:
			IF xOpvEmptied THEN
				iLineStatus:=iLineStatus+1;
			END_IF

		226:
			IF xStackerEmptied THEN
				xLineReady:=TRUE;
			END_IF

	END_CASE

END_ACTION
```

#### LineAlarms.st
```iecst
ACTION LineAlarms:

	//////////////////
	// General Alarms
	//////////////////

	//Reset Alarms//
	IF gMachine.AutoCmd.xReset THEN
		ResetAlarms;
	END_IF

	//Critical//
	//Printer Powered
	IF xLinePoweredON AND NOT Line.Inputs.xPrinterPowered THEN
		Line.Alarms.xAlrPrinterNoPowered := TRUE;
	END_IF

	//Main Supply Overvoltage
	IF NOT Line.Inputs.xOvervoltageProtectionOk THEN
		Line.Alarms.xAlrOvervoltage := TRUE;
	END_IF

	//24VDC Start Sequence Powered
	IF Line.Inputs.x24VdcStartSeqNoPowered THEN
		Line.Alarms.xAlr24VdcStartSeqNoPowered := TRUE;
	END_IF

END_ACTION

ACTION ResetAlarms:
	Line.Alarms := AlarmsReseted;
END_ACTION
```

#### LineAlarmsSummary.st
```iecst
ACTION LineAlarmsSummary:

	//////////////////
	// General Summary
	//////////////////

	//Warnings//
	iReasonWarning.0 := gMachine.AlSummary.xAnyWarning;
	iReasonWarning.1 := Feeder.Alarms.xWarningAlarm;
	iReasonWarning.2 := Primer.Alarms.xWarningAlarm;
	iReasonWarning.3 := Dryer.Alarms.xWarningAlarm;
	iReasonWarning.4 := Stacker.Alarms.xWarningAlarm;
	iReasonWarning.5 := SafetyController.Alarms.xWarningAlarm;
	iReasonWarning.6 := Sarm.Alarms.xWarningAlarm;

	Line.Alarms.xWarningAlarm :=  iReasonWarning > 0;

	//Register the reason of the warning alarm
	IF gMachine.St.Mode.xAuto AND EDGEPOS(Line.Alarms.xWarningAlarm) THEN
		Line.Alarms.iReasonWarning := iReasonWarning;
		LogWarningAlarm;
	ELSIF EDGEPOS(gMachine.St.Mode.xAuto AND NOT Line.Alarms.xWarningAlarm) THEN
		Line.Alarms.iReasonWarning := 0;
	END_IF

	//Alarms stop//
	IF gMachine.AutoCmd.xReset THEN
		iReasonStop := 0;
	END_IF

	IF (Line.Status <> LINE_STOPPED) THEN
		iReasonStop.0 := gMachine.AlSummary.xAlarmStop;
		iReasonStop.1 := Primer.Alarms.xCriticalAlarm;
		iReasonStop.2 := Line.Commands.Stop;
		iReasonStop.3 := CuringLed[1].AlSummary.xAlarmStop;
		iReasonStop.4 := CuringLed[2].AlSummary.xAlarmStop;
		iReasonStop.5 := EdgeHoldDown.AlSummary.xAlarmStop;
		iReasonStop.6 := Sarm.Alarms.xCriticalAlarm;
	END_IF

	Line.Alarms.xStopAlarm :=  iReasonStop > 0;

	//Register the reason of the Stop Alarm
	IF NOT Line.StatusSummary.xControlStopping AND EDGEPOS(Line.Alarms.xStopAlarm) THEN
		Line.Alarms.iReasonStop := iReasonStop;
		LogStopAlarm;
	ELSIF (Line.Status > LINE_STOPPED) THEN
		Line.Alarms.iReasonStop := 0;
	END_IF

	//Critical alarms//
	iReasonCritical.0 := gMachine.AlSummary.xAlarmCritical;
	iReasonCritical.1 := Dryer.Alarms.xCriticalAlarm;
	iReasonCritical.2 := Stacker.Alarms.xCriticalAlarm;
	iReasonCritical.3 := SafetyController.Alarms.xCriticalAlarm;
	iReasonCritical.4 := Line.Alarms.xAlrPrinterNoPowered;
	iReasonCritical.5 := Line.Alarms.xAlrOvervoltage;
	iReasonCritical.6 := Line.Alarms.xAlr24VdcStartSeqNoPowered;
	iReasonCritical.7 := gMachine.In.Buttons.xStop;
	iReasonCritical.8 := OverVarnish.Alarms.xCriticalAlarm;
	iReasonCritical.9 := CuringLed[1].AlSummary.xAlarmCritical;
	iReasonCritical.10 := CuringLed[2].AlSummary.xAlarmCritical;
	iReasonCritical.11 := EdgeHoldDown.AlSummary.xAlarmCritical;

	Line.Alarms.xCriticalAlarm :=  iReasonCritical > 0;

	//Register the reason of the Critical Alarm
	IF gMachine.St.Mode.xAuto AND EDGEPOS(Line.Alarms.xCriticalAlarm) THEN
		Line.Alarms.iReasonCritical := iReasonCritical;
		LogCriticalAlarm;
	ELSIF EDGEPOS(gMachine.St.Mode.xAuto AND NOT Line.Alarms.xCriticalAlarm) THEN
		Line.Alarms.iReasonCritical := 0;
	END_IF

	iReasonResetCondition.0 := (NOT Line.Alarms.xWarningAlarm) AND (Line.Alarms.iReasonWarning > 0);
	iReasonResetCondition.1 := (NOT Line.Alarms.xStopAlarm) AND (Line.Alarms.iReasonStop > 0);
	iReasonResetCondition.2 := (NOT Line.Alarms.xCriticalAlarm) AND (Line.Alarms.iReasonCritical > 0);

	Line.Alarms.xResetCondition :=  iReasonResetCondition > 0;

	xNoAlarmsActive := (NOT Line.Alarms.xCriticalAlarm) AND
						(NOT Line.Alarms.xStopAlarm);

	LightTower;
	SoundLightTower;

END_ACTION
```

#### LineCtrl.st
```iecst
PROGRAM _CYCLIC
	(* Insert code here *)
	Line ACCESS ADR(gLine);
	SafetyController ACCESS ADR (gSafetyController);
	Feeder ACCESS ADR(gFeeder);
	Primer ACCESS ADR(gPrimer);
	Sarm ACCESS ADR(gSarm);
	OverVarnish ACCESS ADR(gOverVarnish);
	Dryer ACCESS ADR(gDryerAnc);
	DryerData ACCESS ADR(gDryerRemoteData);
	Stacker ACCESS ADR(gStacker);
	Machine ACCESS ADR(gMachine);
	Belt ACCESS ADR(gBelt);
	ThickCtrl ACCESS ADR(gThicknessCtrl);
	TransVacuum ACCESS ADR(gTransVacuum);
	CuringLed ACCESS ADR(gCuringLed);
	EdgeHoldDown ACCESS ADR(gEdgeHoldDown);
	BeltClean ACCESS ADR(gBeltClean);

	//Just enter in line if gMachine controlled by line and configured the quantity of external devices
	IF NOT gMachine.Pt.xControlledByLine OR Line.Parameters.iNumExternalDevices = 0 THEN
		RETURN;
	END_IF

	Configuration;

	LineAlarms;

	LineAlarmsSummary;

	xStatusChanged := LineStatusPrevious <> Line.Status;
	IF xStatusChanged THEN xLineReady:=FALSE; iLineStatus:=0; END_IF

	xSubStatusChanged := iLineSubStatusPrevious<>iLineStatus;
	IF xSubStatusChanged THEN LogLineSubStatus;	END_IF

	LineStatusPrevious := Line.Status;
	iLineSubStatusPrevious := iLineStatus;

	//Inputs
	LineInputs;

	//External requests to line from printer (machine) or ancillaries
	LineOrders;

	CASE Line.Status OF

		LINE_NOT_POWERED:
			xLinePoweredON:=FALSE;
			//Waiting the machine to be configured
			IF Line.Parameters.iNumExternalDevices > 0 AND NOT Line.OrdersSw.Shutdown THEN
				Line.Status:=LINE_NOT_INITIALIZED;
			END_IF

		LINE_NOT_INITIALIZED:
			//xLineReady:=FALSE;
			PowerOffLineDevices;
			IF xLinePowered AND xLinePoweredOFF THEN Line.Status:=LINE_INITIALIZING; END_IF

		LINE_POWERING_OFF:
			PowerOffLineDevices;
			IF xLinePoweredOFF THEN Line.Status:=LINE_NOT_POWERED; END_IF

		LINE_INITIALIZING:
			PowerUpLineDevices;
			IF xLineReady AND xLinePoweredON THEN xLineStopped:=TRUE; Line.Status:=LINE_STOPPED; END_IF

		LINE_STOPPED:
			IF gMachine.St.Mode.xAuto THEN
				IF xLineToClean THEN
					xCleanToBeExecuted := TRUE;
					Line.Status:=LINE_PREPARING_CLEANPH;
				ELSIF xLineToCleanBelt THEN
					xCleanBeltToBeExecuted := TRUE;
					Line.Status:=LINE_PREPARING_CLEANBELT;
				ELSIF xNoAlarmsActive THEN
					Line.Status:=LINE_IDLE;
				END_IF
			END_IF

		LINE_IDLE:
			xCleanToBeExecuted:=FALSE;
			xCleanBeltToBeExecuted:=FALSE;
			xPreviousIdle:=TRUE;

			IF Line.OrdersSw.Shutdown THEN
				Line.Status:=LINE_POWERING_OFF;
			END_IF

			IF xLineToPrint AND xNoAlarmsActive THEN
				Line.Status:=LINE_PREPARING_PRINT;
			ELSIF xLineToClean THEN
				xCleanToBeExecuted := TRUE;
				Line.Status:=LINE_PREPARING_CLEANPH;
			ELSIF xLineToCleanBelt AND ThickCtrl.status.Belt.xBeltEmpty THEN
				xCleanBeltToBeExecuted := TRUE;
				Line.Status:=LINE_PREPARING_CLEANBELT;
			ELSIF xLineToEmptyBelt THEN
				Line.Status:=LINE_PREPARING_EMPTYBELT;
			END_IF

		LINE_PREPARING_EMPTYBELT:
			xLineStopped:=FALSE;
			PreparingEmptyBelt;
			IF xLineReady THEN Line.Status:=LINE_STARTING_EMPTYBELT; END_IF

		LINE_STARTING_EMPTYBELT:
			StartingEmptyBelt;
			IF xLineReady THEN Line.Status:=LINE_BELT_EMPTYING; END_IF

		LINE_BELT_EMPTYING:
			//To finish this process automatically when line is full emptied
			EmptyingBelt;
			IF xLineReady THEN Line.Status:=LINE_CONTROLLED_STOP; END_IF

		LINE_PREPARING_PRINT:
			xLineStopped:=FALSE;
			xPreviousPrinting:=FALSE;
			PreparingPrint;
			IF xLineReady THEN Line.Status:=LINE_STARTING_PRINTING; END_IF

		LINE_STARTING_PRINTING:
			StartingPrinting;
			IF xLineReady THEN Line.Status:=LINE_PRINTING; END_IF

		LINE_PRINTING:
			xPreviousIdle:=FALSE;
			IF xLineToPause OR xLineToClean OR xLineToCleanBelt THEN
				IF xLineToClean THEN
					xPreviousPrinting:=TRUE;
					xCleanToBeExecuted := TRUE;
				ELSIF xLineToCleanBelt THEN
					xPreviousPrinting:=TRUE;
					xCleanBeltToBeExecuted := TRUE;
				END_IF
				Line.Status:=LINE_PAUSING;
			END_IF

		LINE_PAUSING:
			xPreviousPausing:=FALSE;
			Pausing;
			IF xLineToClean THEN
				xCleanToBeExecuted := TRUE;
			END_IF

			IF xLineToPrint THEN
				Line.Status:=LINE_PREPARING_PRINT;
			ELSIF xLineReady THEN
				Line.Status:=LINE_PAUSED;
			END_IF

		LINE_PAUSED:
			IF xLineToPrint THEN
				Line.Status:=LINE_PREPARING_PRINT;
			ELSIF xLineToClean THEN
				xCleanToBeExecuted := TRUE;
				xPreviousPausing:=TRUE;
				Line.Status:=LINE_PREPARING_CLEANPH;
			ELSIF xLineToCleanBelt THEN
				xCleanBeltToBeExecuted := TRUE;
				xPreviousPausing:=TRUE;
				Line.Status:=LINE_PREPARING_CLEANBELT;
			END_IF

		LINE_PREPARING_CLEANPH:
			PreparingCleaningPH;
			IF xLineReady THEN Line.Status:=LINE_STARTING_CLEANINGPH; END_IF

		LINE_PREPARING_CLEANBELT:
			PreparingCleaningBelt;
			IF xLineReady THEN Line.Status:=LINE_STARTING_CLEANINGBELT; END_IF

		LINE_STARTING_CLEANINGPH:
			xCleanToBeExecuted := FALSE;
			StartingCleaningPH;
			IF xLineReady THEN Line.Status:=LINE_CLEANINGPH; END_IF

		LINE_STARTING_CLEANINGBELT:
			xCleanBeltToBeExecuted := FALSE;
			StartingCleaningBelt;
			IF xLineReady THEN Line.Status:=LINE_CLEANINGBELT; END_IF

		LINE_CLEANINGPH:
			IF NOT gMachine.St.Position.xCleaning AND NOT BeltClean.Status.xCleaning THEN
				Line.Status:=LINE_CLEANED;
			END_IF

		LINE_CLEANINGBELT:
			CleaningBelt;
			IF xLineReady THEN
				Line.Status:=LINE_CLEANED;
			END_IF

		LINE_CLEANED:
			IF xPreviousPrinting THEN
				Line.Status:=LINE_PREPARING_PRINT;
			ELSIF xPreviousIdle THEN
				Line.Status:=LINE_IDLE;
			ELSIF xPreviousPausing THEN
				Line.Status:=LINE_PAUSING;
			ELSE
				Line.Status:=LINE_STOPPED;
			END_IF

		LINE_CONTROLLED_STOP:
			xCleanBeltToBeExecuted := FALSE;
			ControlStopping;
			IF xLineReady THEN xLineStopped:=TRUE; Line.Status:=LINE_STOPPED; END_IF

		LINE_ERROR:
			Stopping;
			IF xLineReady THEN xLineStopped:=TRUE; Line.Status:=LINE_STOPPED; END_IF

	END_CASE

	StatusSw;
	IF xStatusChanged THEN LogLineSwStatus; END_IF

	//Line state summaries
	IF Line.Status<>LINE_NOT_INITIALIZED AND Line.Status<>LINE_INITIALIZING THEN
		IF NOT (xLinePowered AND xLinePoweredON) THEN
			StopAllLineDevices;
			Line.Status:=LINE_NOT_INITIALIZED;
		ELSIF (NOT xLineStopped) THEN
			IF (NOT gMachine.St.Mode.xAuto) THEN
				Line.Status:=LINE_ERROR;
			ELSIF Line.Alarms.xCriticalAlarm THEN
				Line.Status:=LINE_ERROR;
			ELSIF Line.Alarms.xStopAlarm THEN
				Line.Status:=LINE_CONTROLLED_STOP;
			END_IF
		ELSE
			IF NOT gMachine.St.Mode.xAuto THEN
				Line.Status := LINE_STOPPED;
			END_IF
		END_IF
	END_IF

	//Store the history of the status to easy the debug
	IF Line.Status<>StateHistory[0] THEN
		FOR iIndexHistory:=iHistoryLines TO 1 BY -1 DO
			StateHistory[iIndexHistory]:=StateHistory[iIndexHistory-1];
		END_FOR
		StateHistory[0]:=Line.Status;
	END_IF

	//Previous states
	xFromPause := StateHistory[1] = LINE_PAUSED;

	//Resetting local status variables
	IF EDGEPOS(Line.Alarms.xStopAlarm OR Line.Alarms.xCriticalAlarm) OR Line.StatusSummary.xIdle THEN
		//xPreviousIdle := FALSE;
		xPreviousPausing := FALSE;
		xPreviousPrinting := FALSE;
	END_IF

	//Logging commands
	IF EDGEPOS(Line.Commands.Print) THEN LogPrintCommand; END_IF
	IF EDGEPOS(Line.Commands.Pause) THEN LogPauseCommand; END_IF
	IF EDGEPOS(Line.Commands.Stop) THEN LogStopCommand; END_IF
	IF EDGEPOS(Line.Commands.Clean) THEN LogCleanCommand; END_IF
	IF EDGEPOS(Line.Commands.EmptyBelt) THEN LogEmptyBeltCommand; END_IF

	//Logging buttons
	IF EDGEPOS(gMachine.In.Buttons.xStart) THEN LogStartButton; END_IF
	IF EDGEPOS(gMachine.In.Buttons.xStop) THEN LogStopButton; END_IF

	Line.SubStatus := iLineStatus;

	//Outputs
	LineOutputs;

	//Line commands
	Line.Commands := ResetedLineCommands;

	//Line summary
	Line.StatusSummary.xStopped 		:= Line.Status=LINE_STOPPED OR Line.Status=LINE_IDLE;
	Line.StatusSummary.xErrorStopping 	:= Line.Status=LINE_ERROR;
	Line.StatusSummary.xControlStopping := Line.Status=LINE_CONTROLLED_STOP;
	Line.StatusSummary.xCleaning 		:= (Line.Status=LINE_PREPARING_CLEANPH) OR (Line.Status=LINE_STARTING_CLEANINGPH) OR (Line.Status=LINE_CLEANINGPH) OR (Line.Status=LINE_CLEANED);
	Line.StatusSummary.xCleaningBelt	:= (Line.Status=LINE_PREPARING_CLEANBELT) OR (Line.Status=LINE_STARTING_CLEANINGBELT) OR (Line.Status=LINE_CLEANINGBELT);
	Line.StatusSummary.xPausing 		:= (Line.Status=LINE_PAUSING) OR (Line.Status=LINE_PAUSED);
	Line.StatusSummary.xPrinting 		:= (Line.Status=LINE_PREPARING_PRINT) OR (Line.Status=LINE_STARTING_PRINTING) OR (Line.Status=LINE_PRINTING);
	Line.StatusSummary.xEmptyingBelts 	:= (Line.Status=LINE_PREPARING_EMPTYBELT) OR (Line.Status=LINE_STARTING_EMPTYBELT) OR (Line.Status=LINE_BELT_EMPTYING);
	Line.StatusSummary.xIdle	 		:= Line.Status=LINE_IDLE;

	xFeederEmptied := FeederEmptied(ADR(Feeder));
	xPrimerEmptied := PrimerEmptied(ADR(Primer));
	xSarmEmptied := SarmEmptied(ADR(Sarm));
	xPrinterEmptied := PrinterEmptied(ADR(ThickCtrl));
	xDryerEmptied := DryerEmptied(ADR(Dryer));
	xOpvEmptied := OpvEmptied(ADR(OverVarnish));
	xStackerEmptied := StackerEmptied(ADR(Stacker));
	Line.StatusSummary.xLineEmpty := xFeederEmptied AND xPrimerEmptied AND xSarmEmptied AND xPrinterEmptied AND xDryerEmptied AND xOpvEmptied AND xStackerEmptied; //Status added to let sw know whether line is empty

END_PROGRAM
```

#### LineOrders.st
```iecst
ACTION LineOrders:

	//Line to clean orders
	IF gMachine.St.Cleaning.xCleanRequestToLine THEN
		xCleanRequestToLine := TRUE;
	ELSE
		xCleanRequestToLine := FALSE;
	END_IF

	iReasonLineToClean.0 := Line.Commands.Clean;
	iReasonLineToClean.1 := xCleanRequestToLine;
	iReasonLineToClean.2 := xCleanToBeExecuted;

	xLineToClean := iReasonLineToClean>0;

	iReasonLineToCleanBelt.0 := BeltClean.Status.xCleanRequested;
	iReasonLineToCleanBelt.1 := xCleanBeltToBeExecuted;

	xLineToCleanBelt := iReasonLineToCleanBelt >0 AND gBeltClean.Status.State <> BCLEAN_FAULT;

	IF EdgeHoldDown.status.xEnabled AND (rEhdBarsHeighSp <> EdgeHoldDown.parameters.rBarsHeighSp) THEN
		xEhdRequestToPause := TRUE;

	ELSIF EDGENEG(Line.StatusSummary.xPausing) THEN
		xEhdRequestToPause := FALSE;
	END_IF

	//Line to pause orders
	iReasonLineToPause.0 := Line.Commands.Pause;
	iReasonLineToPause.1 := gMachine.In.Buttons.xStart;
	iReasonLineToPause.2 := Feeder.Alarms.xCriticalAlarm;
	iReasonLineToPause.3 := NOT gMachine.St.xRobotReadyToPrint AND NOT gCamera.OrdersSw.xCalibration;
	iReasonLineToPause.4 := EDGEPOS(xEhdRequestToPause);

	//Saving previous ehd heigh setpoint
	rEhdBarsHeighSp := EdgeHoldDown.parameters.rBarsHeighSp;

	//Line to print orders
	iReasonLineToPrint.0 := Line.Commands.Print;
	iReasonLineToPrint.1 := gMachine.In.Buttons.xStart AND gMachine.St.xRobotReadyToPrint AND Line.Status=LINE_PAUSED;
	iReasonLineToPrint.2 := xEhdRequestToPause AND (EdgeHoldDown.parameters.rBlockPosition>=EdgeHoldDown.status.rBlockPrePrintingPosition) AND Line.Status=LINE_PAUSED; //NOZOMITWO-2420

	//[RGP]DELOREAN-972
	//User request to print
	iReasonRequestLineToPrint.0 := tonLineStartButton.Q AND gMachine.parSw.UI.xStartPrintButtonActive;
	xLineRequestToPrintToSw:=iReasonRequestLineToPrint>0;

	//Empty belt
	iReasonLineToEmptyBelt.0 := Line.Commands.EmptyBelt;

	//To manage that these internal orders are not active at the same time
	IF iReasonLineToPause>0 AND Line.StatusSummary.xPrinting THEN
		xLineToPause := TRUE;

	ELSIF iReasonLineToPrint>0 THEN
		xLineToPrint := TRUE;

	ELSIF iReasonLineToEmptyBelt>0 THEN
		xLineToEmptyBelt := TRUE;

	ELSE
		xLineToPause := FALSE;
		xLineToPrint := FALSE;
		xLineToEmptyBelt := FALSE;
	END_IF

	//EHD
	//To send ehd to resting position when entering idle. So maybe controlled stop has not been executed properly
	IF EDGEPOS(Line.StatusSummary.xIdle) THEN
		EdgeHoldDown.orders.xResetPosition := TRUE;
	ELSIF EdgeHoldDown.status.xInRestingPosition THEN
		EdgeHoldDown.orders.xResetPosition := FALSE;
	END_IF

	//Primer NOZOMITWO-2264
	Primer.Orders.xEnablePriming := NOT Line.StatusSummary.xEmptyingBelts OR NOT Machine.St.HwData.xIsWater;

	//OPV NOZOMITWO-2264
	OverVarnish.Orders.xEnablePriming := NOT Line.StatusSummary.xEmptyingBelts OR NOT Machine.St.HwData.xIsWater;

	//Preprinting position
	ton_FeederEmpty(IN:=(NOT Feeder.Status.Device.xFeeding), PT:=T#20S);
	ton_PrimerBeltEmpty(IN:=((Primer.Inputs.Comms.xBeltEmpty OR NOT Primer.ParSw.xEnabled OR NOT Primer.Parameters.xInstalled) AND Belt.states.xRuningBelt), PT:=T#20S);
	ton_SarmBeltEmpty(IN:=((Sarm.Status.xBeltEmpty OR NOT Sarm.ParSw.xEnabled OR NOT Sarm.Parameters.xInstalled) AND Belt.states.xRuningBelt), PT:=T#20S);

	IF NOT Feeder.ParSw.xEnabled AND NOT Primer.ParSw.xEnabled AND NOT Sarm.ParSw.xEnabled THEN
		//No ancillaries installed before the printer are enabled in remote mode
		Line.Orders.Preprinting := FALSE;

	ELSE
		Line.Orders.Preprinting := 	ton_FeederEmpty.Q AND
									ton_PrimerBeltEmpty.Q AND
									ton_SarmBeltEmpty.Q AND
									(ThickCtrl.status.Belt.xBeltEmpty AND Belt.states.xRuningBelt);
	END_IF

	//SafetyController.Orders.xDisableReadBlock := NOT (gPLC.Internal.Blink_2s.Out AND gPLC.Internal.Blink_1s.Out);
	Feeder.Orders.xDisableReadBlock := NOT (gPLC.Internal.Blink_2s.Out AND gPLC.Internal.Blink_1s.Out) OR NOT Feeder.ParSw.xEnabled;
	Primer.Orders.xDisableReadBlock := NOT (NOT gPLC.Internal.Blink_2s.Out AND gPLC.Internal.Blink_1s.Out) OR NOT Primer.ParSw.xEnabled;
	Sarm.Orders.xDisableReadBlock := NOT (NOT gPLC.Internal.Blink_2s.Out AND gPLC.Internal.Blink_1s.Out) OR NOT Sarm.ParSw.xEnabled;
	OverVarnish.Orders.xDisableReadBlock := NOT (gPLC.Internal.Blink_2s.Out AND NOT gPLC.Internal.Blink_1s.Out) OR NOT OverVarnish.ParSw.xEnabled;
	Stacker.Orders.xDisableReadBlock := NOT (NOT gPLC.Internal.Blink_2s.Out AND NOT gPLC.Internal.Blink_1s.Out) OR NOT Stacker.ParSw.xEnabled;

END_ACTION
```

#### Pausing.st
```iecst
ACTION Pausing:

	IF xStatusChanged THEN
		ton_PrinterBeltInputEmpty.IN := FALSE;
		iLineStatus:=330;
	END_IF

	ton_PrinterBeltInputEmpty();

	CASE iLineStatus OF
		330:
			Feeder.Commands.xPause:=TRUE;
			xFeederPaused := FeederPaused(ADR(Feeder)) OR FeederStopped(ADR(Feeder));
			IF xFeederPaused THEN
				iLineStatus:=iLineStatus+1;
			END_IF

		331:
			Primer.Commands.xPause:=TRUE;
			xPrimerPaused := PrimerPaused(ADR(Primer));
			IF xPrimerPaused THEN
				iLineStatus:=iLineStatus+1;
			END_IF

		332:
			Sarm.Commands.xPause:=TRUE;
			xSarmPaused := SarmPaused(ADR(Sarm));
			IF xSarmPaused THEN
				iLineStatus:=iLineStatus+1;
			END_IF

		333:
			//Timer
			tiTimeToEmpty := REAL_TO_TIME(60 * (gMachine.Pt.CT.rDistanceBeltInitToPd) / Belt.parameters.rSetPointSpeed); //Belt.parameters.rSetPointSpeed minimum value is 5m/min, cannot be 0.
			ton_PrinterBeltInputEmpty.IN := TRUE;
			ton_PrinterBeltInputEmpty.PT := tiTimeToEmpty;

			xPrinterBeltInputEmpty := ton_PrinterBeltInputEmpty.Q;
			IF xPrinterBeltInputEmpty AND xPrinterEmptied THEN
				Dryer.Commands.xPause:=TRUE;
				OverVarnish.Commands.xPause:=TRUE;
				iLineStatus:=iLineStatus+1;
			END_IF

		334:
			xDryerPaused := DryerPaused(ADR(Dryer));
			IF xDryerPaused  THEN
				iLineStatus:=iLineStatus+1;
			END_IF

		335:
			xOverVarnishPaused := OpvPaused(ADR(OverVarnish));
			IF xOverVarnishPaused THEN
				xLineReady:=TRUE;
			END_IF

	END_CASE

END_ACTION
```

#### PowerUpLineDevices.st
```iecst
ACTION PowerUpLineDevices:

	IF xStatusChanged THEN
		iLineStatus:=110;
		iIndexPower:=0;
	END_IF

	CASE iLineStatus OF

		110:
			//Timer
			ton_DelayPowerOn.IN := TRUE;
			ton_DelayPowerOn.PT:= Line.Parameters.ExternalDevices[iIndexPower].tiDelay;
			ton_DelayPowerOn();

			IF Line.Parameters.ExternalDevices[iIndexPower].xIsEngine THEN
				//Activate the first output signal
				Line.Outputs.ExternalDevices[iIndexPower].xOpen:=TRUE;

				IF ton_DelayPowerOn.Q THEN
					//Activate second signal when motorized contactor is loaded
					Line.Outputs.ExternalDevices[iIndexPower].xClose:=TRUE;

					//Go to next
					ResetPowerOnTimerAndNext;
				END_IF

			ELSE
				IF ton_DelayPowerOn.Q THEN
					//Activate both outputs if it is not Motorized contactor
					Line.Outputs.ExternalDevices[iIndexPower].xClose:=TRUE;
					Line.Outputs.ExternalDevices[iIndexPower].xOpen:=TRUE;

					//Go to next
					ResetPowerOnTimerAndNext;
				END_IF
			END_IF
			iLastIndexPower := iIndexPower;

		111:

			IF iIndexPower<=Line.Parameters.iNumExternalDevices THEN
				//If the Index is not the last one, repeate the timer to activate next one
				iLineStatus:=110;
			ELSE
				iLineStatus:=iLineStatus+1;
			END_IF

		112:
			xLinePoweredON := TRUE;
			xLineReady:=TRUE;

	END_CASE

END_ACTION

ACTION ResetPowerOnTimerAndNext:

	//Reset timer
	ton_DelayPowerOn(IN:=FALSE);
	iIndexPower:=iIndexPower+1;
	iLineStatus:=iLineStatus+1;

END_ACTION
```

#### PreparingCleaningBelt.st
```iecst
ACTION PreparingCleaningBelt:

	IF xStatusChanged THEN
		iLineStatus:=700;
	END_IF

	CASE iLineStatus OF
		700:
			IF gBeltClean.Status.State = BCLEAN_FAULT THEN
				xLineReady := TRUE;
			ELSE //IF gThicknessCtrl.status.Belt.xBeltEmpty THEN
				IF xPreviousIdle AND gThicknessCtrl.status.Belt.xBeltEmpty THEN
					gMachine.commands.xRunBelt := TRUE;
				END_IF
				IF gBelt.states.xRuningBelt THEN
					gMachine.commands.CleanBelt.xStart := TRUE;
					xLineReady:=TRUE;
				END_IF
			END_IF

	END_CASE

END_ACTION
```

#### PreparingEmptyBelt.st
```iecst
ACTION PreparingEmptyBelt:

	IF xStatusChanged THEN
		iLineStatus:=200;
	END_IF

	ton_StackerCleanBelts.IN:=Stacker.Outputs.xCleanBelts;
	ton_StackerCleanBelts.PT:=T#2S;
	ton_StackerCleanBelts();

	CASE iLineStatus OF
		200:
			StartBlowers;
			IF ton_StackerCleanBelts.Q OR NOT Stacker.ParSw.xEnabled THEN
				IF (gMachine.St.HwData.xIsWater OR NOT ThickCtrl.status.MediaPosition.xMediaBelowMachine) THEN
					gMachine.commands.xAllToCap := TRUE;
					Stacker.Commands.xPrepare := TRUE;

					xBarsInCapPosition := BarPositionCapped(ADR(Machine));
					IF xBarsInCapPosition THEN iLineStatus:=iLineStatus+1; END_IF

				ELSE
					gMachine.commandsSw.xToNormal_GI := TRUE;
					IF gMachine.St.AutoMode.xProduction THEN
						gMachine.commandsSw.xToNormal_GI := FALSE; //TOREVIEW: This should be an internal command, not something coming from Comms
						gMachine.commands.xAllToPrint:=TRUE;
						Stacker.Commands.xPrepare := TRUE;

						xBarsInPrintingPosition := BarPositionReady(ADR(Machine));
						IF xBarsInPrintingPosition THEN iLineStatus:=iLineStatus+1; END_IF
					END_IF
				END_IF
			END_IF

		201:
			//Waiting stacker and evaluate which next object must be prepared
			xStackerReady := StackerReady(ADR(Stacker));
			IF xStackerReady THEN
				iLineStatus:=iLineStatus+1;
			END_IF

		202:
			OverVarnish.Commands.xPrepare:=TRUE;
			xOverVarnishReady:=OpvReady(ADR(OverVarnish));
			IF xOverVarnishReady THEN
				iLineStatus:=iLineStatus+1;
			END_IF

		203:
			IF (Dryer.ParSw.xEnableArcLamp OR Dryer.ParSw.xEnableNIR) THEN
				Dryer.Commands.xBelEmpty := TRUE;
			ELSE
				Dryer.Commands.xStartTransport:=TRUE;
			END_IF
			iLineStatus:=iLineStatus+1;

		204:
			IF Dryer.Status.CtrlStatus = DRYERCTRL_MOVING AND (Dryer.ParSw.xEnableArcLamp OR Dryer.ParSw.xEnableNIR) THEN
				Dryer.Commands.xPrepare:=TRUE;
			END_IF
			xDryerReady := DryerReady(ADR(Dryer));
			IF xDryerReady THEN xLineReady:=TRUE; END_IF

	END_CASE

END_ACTION

ACTION StartBlowers:
	FOR iIndexTransVacuum:=1 TO MAX_LAST_TRANS_VACUUM DO
		TransVacuum[iIndexTransVacuum].Commands.xRunByLine := TRUE;
	END_FOR
END_ACTION
```

#### StartingEmptyBelt.st
```iecst
ACTION StartingEmptyBelt:

	IF xStatusChanged THEN
		iLineStatus:=210;
	END_IF

	CASE iLineStatus OF
		210:
			Stacker.Commands.xStart:=TRUE;
			iLineStatus:=iLineStatus+1;

		211:
			xStackerStarted:=StackerStarted(ADR(Stacker));
			IF xStackerStarted THEN
				OverVarnish.Commands.xStart:=TRUE;
				iLineStatus:=iLineStatus+1;
			END_IF

		212:
			xOverVarnishStarted:=OpvStarted(ADR(OverVarnish));
			IF xOverVarnishStarted THEN
				Dryer.Commands.xStart:=TRUE;
				iLineStatus:=iLineStatus+1;
			END_IF

		213:
			xDryerStarted:=DryerStarted(ADR(Dryer));
			xThicknessSensorReady := ThicknessSensorReady(ADR(ThickCtrl));
			IF xThicknessSensorReady AND xDryerStarted THEN
				gMachine.commands.xRunBelt := TRUE;
				iLineStatus:=iLineStatus+1;
			END_IF

		214:
			xPrinterBeltStarted:= PrinterBeltStarted(ADR(Belt));
			IF xPrinterBeltStarted THEN
				Sarm.Commands.xStart:=TRUE;
				iLineStatus:=iLineStatus+1;
			END_IF

		215:
			xSarmStarted := SarmStarted(ADR(Sarm));
			IF xSarmStarted THEN
				Primer.Commands.xPrepare:=TRUE;
				iLineStatus:=iLineStatus+1;
			END_IF

		216:
			xPrimerReady:=PrimerReady(ADR(Primer));
			IF xPrimerReady THEN
				Feeder.Commands.xPrepare:=TRUE;
				iLineStatus:=iLineStatus+1;
			END_IF

		217:
			xFeederReady:=FeederReady(ADR(Feeder));
			IF xFeederReady THEN
				xLineReady:=TRUE;
			END_IF

	END_CASE

END_ACTION
```

#### StatusSw.st
```iecst
ACTION StatusSw:
	CASE Line.Status OF
		LINE_NOT_POWERED: Line.StatusSw:= 999;
		LINE_POWERING_OFF: Line.StatusSw:= 60;
		LINE_ERROR:	Line.StatusSw:= 2;
		LINE_PREPARING_EMPTYBELT: Line.StatusSw:= 20;
		LINE_PREPARING_PRINT: Line.StatusSw:= 30;
		LINE_PREPARING_CLEANPH: Line.StatusSw:= 40;
		LINE_PREPARING_CLEANBELT: Line.StatusSw:= 70;
		LINE_STARTING_PRINTING: Line.StatusSw:= 31;
		LINE_STARTING_CLEANINGPH: Line.StatusSw:= 41;
		LINE_STARTING_CLEANINGBELT: Line.StatusSw:= 71;
		LINE_BELT_EMPTYING:	Line.StatusSw:= 22;
		LINE_CLEANED:	Line.StatusSw:= 43;
		LINE_STARTING_EMPTYBELT: Line.StatusSw:= 21;
		LINE_IDLE:	Line.StatusSw:= 11;
		LINE_PRINTING:	Line.StatusSw:= 32;
		LINE_PAUSING:	Line.StatusSw:= 33;
		LINE_PAUSED:	Line.StatusSw:= 34;
		LINE_CLEANINGPH:	Line.StatusSw:= 42;
		LINE_CLEANINGBELT:	Line.StatusSw:= 72;
		LINE_CONTROLLED_STOP:	Line.StatusSw:= 50;
		LINE_STOPPED:	Line.StatusSw:= 10;
		LINE_NOT_INITIALIZED:	Line.StatusSw:= 0;
		LINE_INITIALIZING:	Line.StatusSw:= 5;
	END_CASE

END_ACTION
```

#### SystemsLimits.st
```iecst
FUNCTION FeederMaxMediaWidth
	IF Feeder.ParSw.xEnabled THEN FeederMaxMediaWidth:= Feeder.Parameters.Hw.iMaxMediaWidth; ELSE FeederMaxMediaWidth:= Machine.Pt.Hw.iWidth; END_IF
END_FUNCTION

FUNCTION FeederMaxMediaLength
	IF Feeder.ParSw.xEnabled THEN FeederMaxMediaLength:= Feeder.Parameters.Hw.iMaxMediaLength; ELSE FeederMaxMediaLength:= Machine.parSw.Hw.iMaxMediaLength; END_IF
END_FUNCTION

FUNCTION FeederMaxMediaThickness
	IF Feeder.ParSw.xEnabled THEN FeederMaxMediaThickness:= Feeder.Parameters.Hw.iMaxMediaThickness; ELSE FeederMaxMediaThickness:= REAL_TO_UINT(Machine.Pt.CT.rMaxTicknessMedia*10); END_IF
END_FUNCTION

FUNCTION FeederMinMediaThickness
	IF Feeder.ParSw.xEnabled THEN FeederMinMediaThickness:= Feeder.Parameters.Hw.iMinMediaThickness; ELSE FeederMinMediaThickness:= REAL_TO_UINT(Machine.Pt.CT.rMinTicknessMedia*10); END_IF
END_FUNCTION

FUNCTION FeederMaxSpeed
	IF Feeder.Parameters.xInstalled THEN FeederMaxSpeed:= Feeder.Parameters.Hw.rMaxSpeed; ELSE FeederMaxSpeed:= Belt.states.Hw.rMaxSpeed; END_IF
END_FUNCTION

FUNCTION PrimerMaxMediaWidth
	IF Primer.ParSw.xEnabled THEN PrimerMaxMediaWidth:= Primer.Parameters.Hw.iMaxMediaWidth; ELSE PrimerMaxMediaWidth:= Machine.Pt.Hw.iWidth; END_IF
END_FUNCTION

FUNCTION PrimerMaxMediaLength
	IF Primer.ParSw.xEnabled THEN PrimerMaxMediaLength:= Primer.Parameters.Hw.iMaxMediaLength; ELSE PrimerMaxMediaLength:= Machine.parSw.Hw.iMaxMediaLength; END_IF
END_FUNCTION

FUNCTION PrimerMaxMediaThickness
	IF Primer.ParSw.xEnabled THEN PrimerMaxMediaThickness:= Primer.Parameters.Hw.iMaxMediaThickness; ELSE PrimerMaxMediaThickness:= REAL_TO_UINT(Machine.Pt.CT.rMaxTicknessMedia*10); END_IF
END_FUNCTION

FUNCTION PrimerMinMediaThickness
	IF Primer.ParSw.xEnabled THEN PrimerMinMediaThickness:= Primer.Parameters.Hw.iMinMediaThickness; ELSE PrimerMinMediaThickness:= REAL_TO_UINT(Machine.Pt.CT.rMinTicknessMedia*10); END_IF
END_FUNCTION

FUNCTION PrimerMaxSpeed
	IF Primer.Parameters.xInstalled THEN PrimerMaxSpeed:= Primer.Parameters.Hw.rMaxSpeed; ELSE PrimerMaxSpeed:= Belt.states.Hw.rMaxSpeed; END_IF
END_FUNCTION

FUNCTION DryerMaxMediaWidth
	IF Dryer.ParSw.xEnabled THEN DryerMaxMediaWidth:= Dryer.Parameters.Hw.iMaxMediaWidth; ELSE DryerMaxMediaWidth:= Machine.Pt.Hw.iWidth; END_IF
END_FUNCTION

FUNCTION DryerMaxMediaLength
	IF Dryer.ParSw.xEnabled THEN DryerMaxMediaLength:= Dryer.Parameters.Hw.iMaxMediaLength; ELSE DryerMaxMediaLength:= Machine.parSw.Hw.iMaxMediaLength; END_IF
END_FUNCTION

//FUNCTION DryerMaxMediaThickness
//	IF Dryer.ParSw.xEnabled THEN DryerMaxMediaThickness:= Dryer.Parameters.Hw.iMaxMediaThickness; ELSE DryerMaxMediaThickness:= Machine.Pt.CT.rMaxTicknessMedia*10; END_IF
//END_FUNCTION
//
//FUNCTION DryerMinMediaThickness
//	IF Dryer.ParSw.xEnabled THEN DryerMinMediaThickness:= Dryer.Parameters.Hw.iMinMediaThickness; ELSE DryerMinMediaThickness:= Machine.Pt.CT.rMinTicknessMedia*10; END_IF
//END_FUNCTION

FUNCTION DryerMaxSpeed
	IF Dryer.Parameters.xInstalled THEN DryerMaxSpeed:= Dryer.Parameters.Hw.rMaxSpeed; ELSE DryerMaxSpeed:= Belt.states.Hw.rMaxSpeed; END_IF
END_FUNCTION

FUNCTION OvervarnishMaxMediaWidth
	IF OverVarnish.ParSw.xEnabled THEN OvervarnishMaxMediaWidth:= OverVarnish.Parameters.Hw.iMaxMediaWidth; ELSE OvervarnishMaxMediaWidth:= Machine.Pt.Hw.iWidth; END_IF
END_FUNCTION

FUNCTION OvervarnishMaxMediaLength
	IF OverVarnish.ParSw.xEnabled THEN OvervarnishMaxMediaLength:= OverVarnish.Parameters.Hw.iMaxMediaLength; ELSE OvervarnishMaxMediaLength:= Machine.parSw.Hw.iMaxMediaLength; END_IF
END_FUNCTION

FUNCTION OverVarnishMaxMediaThickness
	IF OverVarnish.ParSw.xEnabled THEN OverVarnishMaxMediaThickness:= OverVarnish.Parameters.Hw.iMaxMediaThickness; ELSE OverVarnishMaxMediaThickness:= REAL_TO_UINT(Machine.Pt.CT.rMaxTicknessMedia*10); END_IF
END_FUNCTION

FUNCTION OverVarnishMinMediaThickness
	IF OverVarnish.ParSw.xEnabled THEN OverVarnishMinMediaThickness:= OverVarnish.Parameters.Hw.iMinMediaThickness; ELSE OverVarnishMinMediaThickness:= REAL_TO_UINT(Machine.Pt.CT.rMinTicknessMedia*10); END_IF
END_FUNCTION

FUNCTION OvervarnishMaxSpeed
	IF OverVarnish.Parameters.xInstalled THEN OvervarnishMaxSpeed:= OverVarnish.Parameters.Hw.rMaxSpeed; ELSE OvervarnishMaxSpeed:= Belt.states.Hw.rMaxSpeed; END_IF
END_FUNCTION

FUNCTION StackerMaxMediaWidth
	IF Stacker.ParSw.xEnabled THEN StackerMaxMediaWidth:= Stacker.Parameters.Hw.iMaxMediaWidth; ELSE StackerMaxMediaWidth:= Machine.Pt.Hw.iWidth; END_IF
END_FUNCTION

FUNCTION StackerMaxMediaLength
	IF Stacker.ParSw.xEnabled THEN StackerMaxMediaLength:= Stacker.Parameters.Hw.iMaxMediaLength; ELSE StackerMaxMediaLength:= Machine.parSw.Hw.iMaxMediaLength; END_IF
END_FUNCTION

FUNCTION StackerMaxMediaThickness
	IF Stacker.ParSw.xEnabled THEN StackerMaxMediaThickness:= Stacker.Parameters.Hw.iMaxMediaThickness; ELSE StackerMaxMediaThickness:= REAL_TO_UINT(Machine.Pt.CT.rMaxTicknessMedia*10); END_IF
END_FUNCTION

FUNCTION StackerMinMediaThickness
	IF Stacker.ParSw.xEnabled THEN StackerMinMediaThickness:= Stacker.Parameters.Hw.iMinMediaThickness; ELSE StackerMinMediaThickness:= REAL_TO_UINT(Machine.Pt.CT.rMinTicknessMedia*10); END_IF
END_FUNCTION

FUNCTION StackerMaxSpeed
	IF Stacker.Parameters.xInstalled THEN StackerMaxSpeed:= Stacker.Parameters.Hw.rMaxSpeed; ELSE StackerMaxSpeed:= Belt.states.Hw.rMaxSpeed; END_IF
END_FUNCTION

FUNCTION SarmMaxMediaWidth
	IF Sarm.ParSw.xEnabled THEN SarmMaxMediaWidth:= Sarm.Parameters.Hw.iMaxMediaWidth; ELSE SarmMaxMediaWidth:= Machine.Pt.Hw.iWidth; END_IF
END_FUNCTION

FUNCTION SarmMaxMediaLength
	IF Sarm.ParSw.xEnabled THEN SarmMaxMediaLength:= Sarm.Parameters.Hw.iMaxMediaLength; ELSE SarmMaxMediaLength:= Machine.parSw.Hw.iMaxMediaLength; END_IF
END_FUNCTION

FUNCTION SarmMaxMediaThickness
	IF Sarm.ParSw.xEnabled THEN SarmMaxMediaThickness:= Sarm.Parameters.Hw.iMaxMediaThickness; ELSE SarmMaxMediaThickness:= REAL_TO_UINT(Machine.Pt.CT.rMaxTicknessMedia*10); END_IF
END_FUNCTION

FUNCTION SarmMinMediaThickness
	IF Sarm.ParSw.xEnabled THEN SarmMinMediaThickness:= Sarm.Parameters.Hw.iMinMediaThickness; ELSE SarmMinMediaThickness:= REAL_TO_UINT(Machine.Pt.CT.rMinTicknessMedia*10); END_IF
END_FUNCTION

FUNCTION SarmMaxSpeed
	IF Sarm.Parameters.xInstalled THEN SarmMaxSpeed:= Sarm.Parameters.Hw.rMaxSpeed; ELSE SarmMaxSpeed:= Belt.states.Hw.rMaxSpeed; END_IF
END_FUNCTION
```

#### SystemsReady.st
```iecst
(* TODO: Add your comment here *)
FUNCTION CuringSystemsReady
	//TODO: Implement
	CuringSystemsReady:= CuringLed.Status.State = CURINGLED_READY OR NOT CuringLed.Parameters.xEnabled;
END_FUNCTION

(* Return if the bars are in Position ready to print *)
FUNCTION JobReady
	JobReady := Machine.St.xRobotReadyToPrint ;
END_FUNCTION

(* Return if the bars are in Position ready to print *)
FUNCTION BarPositionReady
	BarPositionReady := Machine.St.Position.xInPrint;
END_FUNCTION

(* Return if the bars are in Position ready to print *)
FUNCTION BarPositionCapped
	BarPositionCapped := Machine.St.Position.xInCap;
END_FUNCTION

(* Return if the bars are in Position ready to print *)
FUNCTION BarPositionCleaning
	BarPositionCleaning := Machine.St.Position.xCleaning;
END_FUNCTION

(* TODO: Add your comment here *)
FUNCTION FeederReady
	FeederReady:= NOT Feeder.ParSw.xEnabled OR NOT Feeder.Parameters.xInstalled OR Feeder.Status.CtrlStatus = FEEDERCTRL_PREPARED OR Feeder.Status.CtrlStatus = FEEDERCTRL_PAUSED;
END_FUNCTION

(* TODO: Add your comment here *)
FUNCTION PrimerReady
	PrimerReady:= NOT Primer.ParSw.xEnabled OR NOT Primer.Parameters.xInstalled OR Primer.Status.CtrlStatus = PRIMERCTRL_PREPARED OR Primer.Status.CtrlStatus = PRIMERCTRL_PAUSED;
END_FUNCTION

(* TODO: Add your comment here *)
FUNCTION SarmReady
	SarmReady:= NOT Sarm.ParSw.xEnabled OR NOT Sarm.Parameters.xInstalled OR Sarm.Status.CtrlStatus = SARMCTRL_STOPPED;
END_FUNCTION

(* TODO: Add your comment here *)
FUNCTION DryerReady
	DryerReady:= NOT Dryer.ParSw.xEnabled OR NOT Dryer.Parameters.xInstalled OR Dryer.Status.CtrlStatus = DRYERCTRL_PREPARED OR Dryer.Status.CtrlStatus = DRYERCTRL_PAUSED OR Dryer.Status.CtrlStatus = DRYERCTRL_DRYING OR (Dryer.Status.CtrlStatus = DRYERCTRL_MOVING AND NOT (Dryer.ParSw.xEnableArcLamp OR Dryer.ParSw.xEnableNIR));
END_FUNCTION

(* TODO: Add your comment here *)
FUNCTION OpvReady
	OpvReady:= NOT OverVarnish.ParSw.xEnabled OR NOT OverVarnish.Parameters.xInstalled OR OverVarnish.Status.CtrlStatus = OPVCTRL_PREPARED OR OverVarnish.Status.CtrlStatus = OPVCTRL_PAUSED;
END_FUNCTION

(* TODO: Add your comment here *)
FUNCTION StackerReady
	StackerReady:=NOT Stacker.ParSw.xEnabled OR NOT Stacker.Parameters.xInstalled OR Stacker.Status.CtrlStatus = STACKERCTRL_PREPARED OR Stacker.Status.CtrlStatus = STACKERCTRL_WORKING;
END_FUNCTION

(* TODO: Add your comment here *)
FUNCTION EhdReady
	EhdReady:= NOT EdgeHoldDown.parSw.xEnable OR NOT EdgeHoldDown.parameters.xInstalled OR EdgeHoldDown.status.xInRestingPosition;
END_FUNCTION

FUNCTION EhdAdjusted
	EhdAdjusted:= NOT EdgeHoldDown.parSw.xEnable OR NOT EdgeHoldDown.parameters.xInstalled OR EdgeHoldDown.status.xAdjustedToMedia;
END_FUNCTION
```

#### SystemsStarted.st
```iecst
(* TODO: Add your comment here *)
FUNCTION FeederStarted
	FeederStarted:= NOT Feeder.ParSw.xEnabled OR NOT Feeder.Parameters.xInstalled OR Feeder.Status.CtrlStatus = FEEDERCTRL_STARTING OR Feeder.Status.CtrlStatus = FEEDERCTRL_FEEDING;
END_FUNCTION

(* TODO: Add your comment here *)
FUNCTION PrimerStarted
	PrimerStarted:= NOT Primer.ParSw.xEnabled OR NOT Primer.Parameters.xInstalled OR Primer.Status.CtrlStatus = PRIMERCTRL_WORKING;
END_FUNCTION

(* TODO: Add your comment here *)
FUNCTION SarmStarted
	SarmStarted:= NOT Sarm.ParSw.xEnabled OR NOT Sarm.Parameters.xInstalled OR Sarm.Status.CtrlStatus = SARMCTRL_RUNNING;
END_FUNCTION

(* TODO: Add your comment here *)
FUNCTION DryerStarted
	DryerStarted:= NOT Dryer.ParSw.xEnabled OR NOT Dryer.Parameters.xInstalled OR Dryer.Status.CtrlStatus = DRYERCTRL_DRYING OR (Dryer.Status.CtrlStatus = DRYERCTRL_MOVING AND NOT (Dryer.ParSw.xEnableArcLamp OR Dryer.ParSw.xEnableNIR));
END_FUNCTION

(* TODO: Add your comment here *)
FUNCTION OpvStarted
	OpvStarted:= NOT OverVarnish.ParSw.xEnabled OR NOT OverVarnish.Parameters.xInstalled OR OverVarnish.Status.CtrlStatus = OPVCTRL_WORKING;
END_FUNCTION

(* TODO: Add your comment here *)
FUNCTION StackerStarted
	StackerStarted:=NOT Stacker.ParSw.xEnabled OR NOT Stacker.Parameters.xInstalled OR Stacker.Status.CtrlStatus = STACKERCTRL_WORKING;
END_FUNCTION

(* TODO: Add your comment here *)
FUNCTION ThicknessSensorReady
	ThicknessSensorReady := ThickCtrl.status.DetectionSystem.xInPosition;
END_FUNCTION

(* TODO: Add your comment here *)
FUNCTION PrinterBeltStarted
	PrinterBeltStarted:=Belt.states.xRuningBelt;
END_FUNCTION

(* TODO: Add your comment here *)
FUNCTION CuringSystemsStarted
	//TODO: Implement
	CuringSystemsStarted:= CuringLed.Status.State = CURINGLED_EMITTING;
END_FUNCTION
```

### Package Logical/Printer - Main project P4 based on refactoring

### BlockInputsMapping.var
```iecst
VAR
	iIndexBlockIn : USINT;
	iIndexJam : USINT;
	dataJam : REFERENCE TO JamDetect_typ;
END_VAR
```

### Program Logical/Printer/BlockSignalsManager/BlockOutputsMapping (IEC)

#### BlockOutputsMapping.st - Init, cyclic, exit code
```iecst
PROGRAM _CYCLIC

	FOR iIndexBlock:=GC_FIRST_BLOCK TO gMachine.Pt.CT.iNumBlocks DO
		// gBlockOutputs is stBlock_Outputs: Used for mapping physical outputs block to logical block
		gBlockOutputs[gBlock[iIndexBlock].parameters.iMappingBlock]:= gBlock[iIndexBlock].Out;

	END_FOR;

	//////////////////////////////////////////
	// JAM OUTPUTS ASSIGNATION
	IF NOT gMachine.parSw.xJamDetectEnable THEN
		RETURN;
	END_IF

	FOR iIndexJam:=1 TO gMachine.St.iJamDevices DO

		//Reference working data to the general data
		dataJam ACCESS ADR(gJamDetect[iIndexJam]);

		IF dataJam.Parameters.iMappingJam > 0 AND dataJam.Parameters.iMappingJam <= MAX_LAST_JAMDEVICE THEN
			gJamOutputs[dataJam.Parameters.iMappingJam] := dataJam.Outputs;
		END_IF

	END_FOR;

END_PROGRAM
```

#### BlockOutputsMapping.var - Local variables
```iecst
VAR
	iIndexBlock : USINT;
	iIndexJam : USINT;
	dataJam : REFERENCE TO JamDetect_typ;
END_VAR
```

### Program Logical/Printer/Config/MachineConfigurator (IEC)

#### MachineConfigurator.st - Init, cyclic, exit code
```iecst
PROGRAM _INIT
	// Safety Visu named Panel needs this variable. It is showing has is configured
	//SAFETY g_xInputSelectMachine;
	g_xInputSelectMachine;

END_PROGRAM

PROGRAM _CYCLIC

	////////////////////////////////////////////////////////////////////////////////////////////////////////////
	// GENERAL
	////////////////////////////////////////////////////////////////////////////////////////////////////////////

	MachineModel;

	//Determine number of last block
	CASE gMachine.Pt.MachineModel OF

		Type_P4_12B_L,
		Type_P4_12B:
			gMachine.Pt.CT.iNumBlocks:=2;
			gMachine.Pt.CT.iNumTransVacuum := 0;
			gMachine.Pt.xControlledByLine := FALSE;

		Type_P4_6B_L,
		Type_P4_6B,
		Type_P4_CBK,
		Type_SHLD,
		Type_S1400,
		Type_P5_OIL,
		Type_P5_WTR:
			gMachine.Pt.CT.iNumBlocks:=1;
			gMachine.Pt.CT.iNumTransVacuum := 0;
			gMachine.Pt.xControlledByLine := FALSE;

		Type_S1400_VAC_PWRLNK,
		Type_S1400_VAC_CAN:
			gMachine.Pt.CT.iNumBlocks:=1;
			gMachine.Pt.CT.iNumTransVacuum := 2;
			gMachine.Pt.xControlledByLine := FALSE;

		Type_NOZ_2_AQ,
		Type_NOZ_2_UV,
		Type_NOZ_2_UV_White,
		Type_MECANO_UV_WHITE,
		Type_MECANO_UV_OPV,
		Type_MECANO_UV_WHITE_OPV:
			gMachine.Pt.CT.iNumBlocks:=1;
			gMachine.Pt.CT.iNumTransVacuum := 2;
			gMachine.Pt.xControlledByLine := TRUE;

		Type_CUBE,
		Type_CUBE_INSPECTION,
		Type_CUBE_GULLIVER,
		Type_CUBE_GULLIVER_INSPECTION:
			gMachine.Pt.CT.iNumBlocks:=1;
			gMachine.Pt.CT.iNumTransVacuum := 1;
			gMachine.Pt.xControlledByLine := FALSE;

	END_CASE

	//Determine machine direction
	// RIGHT: gMachine.parSw.xMachineDirection is 0 or FALSE
	// LEFT:  gMachine.parSw.xMachineDirection is 1 or TRUE
	gMachine.Pt.xLeftHandMachine := gMachine.parSw.xMachineDirection;
	gMachine.Pt.xRightHandMachine:= NOT gMachine.Pt.xLeftHandMachine;

	AsignCommonData;

	CASE gMachine.Pt.ConfigNameID OF

		GC_CONFIG_2BK12BAR_ID:
			AsignDataP4;

		GC_CONFIG_1BK2BAR_ID:
			AsignDataShld;

		GC_CONFIG_BM_1BK8BAR_ID:
			CASE gMachine.Pt.MachineModel OF
				Type_S1400,
				Type_P5_OIL,
				Type_P5_WTR:
					AsignDataP5;
					Type_S1400_VAC_PWRLNK,
				Type_S1400_VAC_CAN:
					AsignDataS1400;
			END_CASE

		GC_CONFIG_1BK8BAR_NOZ2_ID:
			CASE gMachine.Pt.MachineModel OF
				Type_NOZ_2_AQ,
				Type_NOZ_2_UV,
				Type_NOZ_2_UV_White:
					AsignDataNozomi2;
			END_CASE

		GC_CONFIG_1BK8BAR_NOZ2_AQ_ID:
			CASE gMachine.Pt.MachineModel OF
				Type_NOZ_2_AQ:
				AsignDataNozomi2;
			END_CASE

		GC_CONFIG_1BK7BAR_CUBE_ID:
			CASE gMachine.Pt.MachineModel OF
				Type_CUBE,
				Type_CUBE_INSPECTION,
				Type_CUBE_GULLIVER,
				Type_CUBE_GULLIVER_INSPECTION:
					AsignDataCube;
			END_CASE

		GC_CONFIG_1BK10BAR_MECANO_ID:
			CASE gMachine.Pt.MachineModel OF
				Type_MECANO_UV_WHITE,
				Type_MECANO_UV_OPV,
				Type_MECANO_UV_WHITE_OPV:
					AssignDataMecano;
			END_CASE

		GC_CONFIG_PLCDIAGNOSIS_ID:
			AsignDataPlcDiagnosis;

		GC_CONFIG_SIMTEST_ID:

			CASE gSimMachine.Parameters.MachineType OF
				SIM_MACHINE_2B12BAR,
				SIM_MACHINE_1B6BAR,
				SIM_MACHINE_P4_CBK:
					AsignDataP4;

				SIM_MACHINE_1B2BAR:
					AsignDataShld;

				SIM_MACHINE_S1400_VAC_PWRLNK,
				SIM_MACHINE_S1400_VAC_CAN:
					AsignDataS1400;

				SIM_MACHINE_P5_WAT:
					AsignDataP5;

				SIM_MACHINE_NZ2,
				SIM_MACHINE_NZ2_UV,
				SIM_MACHINE_NZ2_UV_WHITE:
					AsignDataNozomi2;

				SIM_MACHINE_CUBE,
				SIM_MACHINE_CUBE_GULLIVER:
					AsignDataCube;

				SIM_MACHINE_MECANO_UV_WHITE,
				SIM_MACHINE_MECANO_UV_OPV,
				SIM_MACHINE_MECANO_UV_WHITE_OPV:
					AssignDataMecano;

			END_CASE
	END_CASE

	JamVibrationConfiguration;

	FOR iBlockIndex:=GC_FIRST_BLOCK TO gMachine.Pt.CT.iNumBlocks DO

		IF gMachine.In.Buttons.xReset THEN
			gBlock[iBlockIndex].Out.xEnableDrive:= TRUE;
			gBlock[iBlockIndex].Out.xEnableIclaSI:= TRUE;
		END_IF

		// Enable Drive AND Icla_SI BK
		IF gMachine.In.Buttons.xZero OR
			(NOT gBlock[iBlockIndex].parSw.xEnableToMovements) THEN
			gBlock[iBlockIndex].Out.xEnableDrive:= FALSE;
			gBlock[iBlockIndex].Out.xEnableIclaSI:= FALSE;
		END_IF

	END_FOR

	MachineModelCopy := gMachine.Pt.MachineModel;

END_PROGRAM
```

#### InputsMachineModel.st - Inputs to determine MachineModel by codification
```iecst
ACTION InputsMachineModel:

	CASE gMachine.Pt.ConfigNameID OF

		GC_CONFIG_2BK12BAR_ID:
			gMachine.In.iMachineModelCode.5:= X20DIF371_003.DInput[2]; (*DI1*)
			gMachine.In.iMachineModelCode.4:= X20DIF371_003.DInput[3]; (*DI2*)
			gMachine.In.iMachineModelCode.3:= X20DIF371_003.DInput[4]; (*DI3*)
			gMachine.In.iMachineModelCode.2:= X20DIF371_003.DInput[5]; (*DI4*)
			gMachine.In.iMachineModelCode.1:= X20DIF371_003.DInput[6]; (*DI6*)
			gMachine.In.iMachineModelCode.0:= X20DIF371_003.DInput[7]; (*DI6*)

		GC_CONFIG_1BK2BAR_ID:
			gMachine.In.iMachineModelCode.3 	:= X20DIF371_002.DInput[11];
			gMachine.In.iMachineModelCode.2 	:= X20DIF371_002.DInput[12];
			gMachine.In.iMachineModelCode.1 	:= X20DIF371_002.DInput[13];
			gMachine.In.iMachineModelCode.0 	:= X20DIF371_002.DInput[14];

		GC_CONFIG_BM_1BK8BAR_ID:
			gMachine.In.iMachineModelCode.0		:= X20DIF371_001.DInput[1];
			gMachine.In.iMachineModelCode.1		:= X20DIF371_001.DInput[2];
			gMachine.In.iMachineModelCode.2		:= X20DIF371_001.DInput[3];
			gMachine.In.iMachineModelCode.3		:= X20DIF371_001.DInput[4];
			gMachine.In.iMachineModelCode.4		:= X20DIF371_001.DInput[5];
			gMachine.In.iMachineModelCode.5		:= X20DIF371_001.DInput[6];

		GC_CONFIG_1BK8BAR_NOZ2_ID,
		GC_CONFIG_1BK8BAR_NOZ2_AQ_ID,
		GC_CONFIG_1BK7BAR_CUBE_ID,
		GC_CONFIG_1BK10BAR_MECANO_ID:
			gMachine.In.iMachineModelCode.0			:= Pdc_X20DIF371_002.DInput[1];
			gMachine.In.iMachineModelCode.1			:= Pdc_X20DIF371_002.DInput[2];
			gMachine.In.iMachineModelCode.2			:= Pdc_X20DIF371_002.DInput[3];
			gMachine.In.iMachineModelCode.3			:= Pdc_X20DIF371_002.DInput[4];
			gMachine.In.iMachineModelCode.4			:= Pdc_X20DIF371_002.DInput[5];
			gMachine.In.iMachineModelCode.5			:= Pdc_X20DIF371_002.DInput[6];

	END_CASE

END_ACTION
```
